Yaskawa INFORM job: X2_57-69(2)(90,180)_HARDOX.JBI

/JOB
//NAME X2_57-69(2)(90,180)_HARDOX
//POS
///NPOS 751,751,751,36,0,0
///TOOL 0
///POSTYPE PULSE
///PULSE
C00000=2000,-108350,-112464,0,80055,0
C00001=-117728,-108350,-112464,-34609,80055,-28580
C00002=-124329,53851,34766,-36826,59228,-24303
C00003=-132418,78233,54919,-18007,48363,-36393
C00004=-132091,87021,68515,-19398,44781,-35491
C00005=-131964,91219,74916,-20112,43130,-35046
C00006=-131964,92220,77875,-20603,41902,-34745
C00007=-131925,92203,77341,-20509,42211,-34802
C00008=-131397,96741,83157,-21411,41178,-34254
C00009=-131925,92203,77341,-20509,42211,-34802
C00010=-132378,78684,56627,-18262,47592,-36223
C00011=-132682,70057,46287,-17529,49367,-36706
C00012=-119143,48210,55676,-30149,44593,20608
C00013=-119357,47156,53956,-26116,42767,17551
C00014=-120340,57080,66927,-26977,39866,17985
C00015=-120719,61633,72965,-27509,38514,18256
C00016=-120718,63903,77470,-28475,37088,18806
C00017=-120500,60851,73214,-27972,38091,18544
C00018=-120914,65321,78494,-28289,37111,18678
C00019=-120500,60851,73214,-27972,38091,18544
C00020=-119122,46332,54187,-26526,42331,17820
C00021=-118999,38480,45168,-29507,46176,20252
C00022=-119368,-115903,-71302,-26914,50601,18610
C00023=-64607,-7982,-59747,18064,104585,-18556
C00024=-122585,1659,-29054,-2148,106745,-41963
C00025=-124057,3295,-23736,-2114,104277,-42416
C00026=-123367,1653,-22955,-2102,102971,-42158
C00027=-123367,1653,-22955,-2102,102971,-42158
C00028=-123367,1464,-21676,-2095,102091,-42146
C00029=-123367,1491,-21879,-2095,102231,-42148
C00030=-122595,1438,-21925,-2097,102251,-41888
C00031=-123098,1579,-22644,-2101,102754,-42066
C00032=-121099,-5117,-28172,-2107,102765,-41388
C00033=-121099,-5224,-27431,-2104,102256,-41380
C00034=-121096,-3542,-26064,-2104,102281,-41379
C00035=-121100,-4913,-29379,-2118,103615,-41403
C00036=-122679,50337,23961,-2073,99143,-41860
C00037=-122679,50327,24372,-2073,98885,-41856
C00038=-122679,50317,25468,-2068,98206,-41845
C00039=-122679,50317,25291,-2069,98316,-41847
C00040=-122229,50284,25254,-2070,98333,-41695
C00041=-122585,50333,23899,-2075,99182,-41830
C00042=-123436,20127,-8164,-2111,103367,-42191
C00043=-123085,19869,-6825,-2101,102422,-42055
C00044=-123085,19731,-5772,-2095,101704,-42044
C00045=-123090,19755,-5955,-2095,101829,-42046
C00046=-122355,19706,-6001,-2097,101852,-41798
C00047=-123021,19907,-7099,-2102,102614,-42036
C00048=-119603,42824,-10224,-2319,104332,-40939
C00049=-124323,33374,-11816,19552,90115,-11471
C00050=-119580,38024,-5833,18417,96098,-9015
C00051=-118818,47331,4592,18589,99387,-8235
C00052=-118854,51639,9991,18809,101216,-7946
C00053=-118854,51688,9891,18816,101298,-7933
C00054=-118396,53981,12432,18736,100835,-7852
C00055=-118854,51688,9891,18816,101298,-7933
C00056=-118058,50558,8647,18739,101302,-7659
C00057=-117672,49987,8022,18702,101306,-7525
C00058=-118854,52185,8952,18883,102088,-7807
C00059=-119377,80940,37276,19231,105085,60834
C00060=-119383,81426,41090,19027,103098,60507
C00061=-119383,81149,41970,18967,102452,60403
C00062=-119503,81114,41806,19281,102559,60100
C00063=-121982,78312,38330,19114,103772,59696
C00064=-119503,81115,41806,19281,102559,60100
C00065=-119566,48683,6206,18410,91622,58331
C00066=-120090,49584,7189,18533,91599,58154
C00067=-122107,80076,35944,19363,106046,60027
C00068=-125220,60788,2341,21151,116877,60889
C00069=-125220,60788,2341,21151,116877,60889
C00070=-126916,76750,29022,19801,109531,58906
C00071=-127645,78004,33974,19502,107427,58282
C00072=-127487,77220,34582,19410,106657,58208
C00073=-127487,77257,34498,19419,106724,58220
C00074=-127913,74998,31769,19485,107311,58167
C00075=-127487,77257,34498,19419,106724,58220
C00076=-124885,43382,-3109,13584,94897,56190
C00077=-125658,44980,-1455,13763,94829,55937
C00078=-126891,66473,19769,17526,104309,57625
C00079=-124484,22564,-21459,18200,86590,59420
C00080=-124478,22213,-20236,18209,85701,59290
C00081=-124478,22285,-20344,18209,85798,59305
C00082=-123939,24375,-18336,18026,85535,59441
C00083=-124479,22285,-20344,18209,85798,59305
C00084=-127548,40111,-4274,24755,95305,61297
C00085=-126910,38918,-5604,24621,95320,61520
C00086=-125531,30039,-16063,20855,91192,60400
C00087=-110493,47386,-4176,13132,86201,63779
C00088=-94830,35895,-16474,7059,86110,68517
C00089=-90477,52028,10631,17758,71006,71149
C00090=-89713,50542,11420,17514,69656,71213
C00091=-89905,50195,13035,17735,68577,70980
C00092=-89905,50233,12920,17724,68663,70994
C00093=-89883,52518,15431,17756,68305,70946
C00094=-89905,50233,12920,17724,68663,70994
C00095=-89391,49561,12188,17458,68659,71180
C00096=-88735,49652,12286,17139,68513,71391
C00097=-89905,50707,11616,17609,69662,71147
C00098=-93822,108273,63701,18536,93326,72680
C00099=-93822,107828,64715,18513,92516,72556
C00100=-93690,107878,66461,18471,91489,72445
C00101=-93690,107926,66303,18474,91606,72462
C00102=-93713,104164,61367,18504,92662,72614
C00103=-93690,107926,66303,18474,91606,72462
C00104=-88166,79692,31239,6097,86382,71862
C00105=-88845,80022,31647,6308,86349,71646
C00106=-88428,80564,30105,6176,87540,71836
C00107=-94090,77517,21608,6175,108524,71897
C00108=-94073,76835,21790,6154,108061,71879
C00109=-94073,75515,22880,6101,106718,71810
C00110=-94073,75604,22800,6105,106813,71815
C00111=-94282,72960,19602,6147,107436,71779
C00112=-94073,75604,22800,6105,106813,71815
C00113=-90523,44446,-9492,-1446,93970,71247
C00114=-91337,44548,-9384,-1199,93942,71004
C00115=-92199,55185,-1301,1007,99713,71206
C00116=-93265,18749,-25601,10213,78649,72540
C00117=-93039,18272,-23901,10154,77351,72504
C00118=-93006,18125,-22740,10166,76573,72452
C00119=-93006,18220,-22895,10161,76715,72464
C00120=-92959,20732,-20534,10144,76549,72465
C00121=-93006,18220,-22895,10161,76715,72464
C00122=-92400,18138,-22970,9886,76649,72654
C00123=-91733,17968,-23126,9585,76586,72864
C00124=-92687,19123,-24402,9968,78051,72675
C00125=-105388,2298,-39102,15529,80254,68873
C00126=-105388,1873,-38509,15552,79692,68802
C00127=-105388,1357,-37735,15585,78976,68710
C00128=-105388,1531,-38004,15573,79223,68742
C00129=-105945,-2529,-41383,15810,79315,68575
C00130=-105945,-2767,-41013,15826,78977,68531
C00131=-105742,-504,-39143,15739,78954,68594
C00132=-105548,-1447,-42806,15582,80627,68872
C00133=-86161,-6758,-47097,6979,78098,74729
C00134=-86311,-6793,-45530,7072,77135,74626
C00135=-86311,-7203,-44912,7084,76549,74590
C00136=-86311,-7084,-45095,7079,76721,74599
C00137=-86468,-10850,-48057,7154,76621,74544
C00138=-86468,-11058,-47732,7163,76316,74526
C00139=-86253,-9013,-46134,7061,76366,74599
C00140=-85946,-9538,-48533,6889,77540,74761
C00141=-91638,-28469,-60972,19623,77269,75627
C00142=-91723,-28440,-59926,19705,76695,75503
C00143=-91723,-28859,-59144,19755,76040,75393
C00144=-91723,-28693,-59463,19734,76307,75438
C00145=-94312,-27181,-58426,20833,77031,74680
C00146=-94312,-27381,-58052,20856,76717,74626
C00147=-93375,-28035,-58503,20460,76442,74902
C00148=-94102,-28107,-59801,20714,77326,74807
C00149=-75235,-25991,-61706,17727,76646,82454
C00150=-74355,-27115,-59920,17436,74870,82487
C00151=-74355,-27621,-59040,17497,74104,82374
C00152=-74355,-27526,-59211,17485,74251,82396
C00153=-73057,-27237,-59013,16875,74023,82799
C00154=-74355,-27526,-59211,17485,74251,82396
C00155=-77057,-4626,-46977,21243,91479,85327
C00156=-76984,-7096,-48960,21220,91416,85338
C00157=-74796,-23928,-59379,17950,77960,82962
C00158=-62955,11917,-39245,-2282,95516,82905
C00159=-62775,11091,-38612,-2332,94707,82971
C00160=-62775,10339,-37928,-2329,93898,82983
C00161=-62775,10494,-38073,-2330,94067,82980
C00162=-63812,9884,-38615,-2013,94064,82672
C00163=-62775,10494,-38073,-2330,94067,82980
C00164=-63124,13025,-35796,-2226,93958,82878
C00165=-62775,11512,-38975,-2336,95146,82960
C00166=-85068,-3435,-45765,9377,101067,77801
C00167=-80917,-22804,-55283,8465,96602,78792
C00168=-82338,-24881,-56282,8726,96296,78315
C00169=-82338,-25559,-54893,8703,95107,78232
C00170=-82338,-25498,-55026,8705,95219,78240
C00171=-82456,-28244,-56927,8723,94993,78185
C00172=-82338,-25498,-55026,8705,95219,78240
C00173=-82992,-25583,-55084,8828,95278,78035
C00174=-84316,-25471,-55005,9073,95425,77617
C00175=-82338,-24922,-56206,8726,96230,78312
C00176=-65428,-70038,-75520,-7958,62422,82819
C00177=-65283,-69785,-73717,-8103,61466,82944
C00178=-65283,-69734,-72466,-8160,60731,82996
C00179=-65283,-69744,-72637,-8152,60830,82990
C00180=-65562,-66708,-71125,-7963,61427,82841
C00181=-65283,-69745,-72637,-8152,60830,82990
C00182=-76204,-68518,-72352,8123,61758,80129
C00183=-74993,-68244,-72242,7504,61717,80585
C00184=-69704,-69532,-74690,-998,61942,81859
C00185=-78060,-84536,-88579,-1407,62283,78117
C00186=-78060,-84536,-88579,-1407,62283,78117
C00187=-64607,-7982,-59747,18064,104585,-18556
C00188=-43259,-142284,-94849,-68481,67043,-45987
C00189=-75789,-57542,-35879,-68380,64193,-60275
C00190=-79378,-55423,-31936,-68889,61283,-60160
C00191=-80801,-54484,-30299,-69115,60133,-60112
C00192=-80803,-53463,-27973,-69597,59790,-59668
C00193=-80780,-53792,-28606,-69479,59888,-59772
C00194=-82380,-55228,-29381,-69587,58724,-59873
C00195=-80801,-53699,-28530,-69478,59874,-59776
C00196=-81788,-51404,-27272,-69234,59369,-60118
C00197=-80801,-53699,-28530,-69478,59874,-59776
C00198=-79378,-54655,-30185,-69233,61022,-59829
C00199=-75790,-56818,-34168,-68680,63927,-59955
C00200=-84853,-69188,-42023,-59966,34850,-64425
C00201=-87616,-64026,-36454,-59770,32751,-64733
C00202=-88672,-61932,-34175,-59731,31934,-64834
C00203=-88674,-60834,-31833,-60968,31481,-64183
C00204=-88651,-60985,-32132,-60826,31549,-64256
C00205=-90372,-59623,-31443,-59618,30637,-65026
C00206=-88651,-60985,-32132,-60826,31549,-64256
C00207=-87595,-63088,-34428,-60823,32369,-64172
C00208=-84831,-68269,-40036,-60922,34477,-63902
C00209=-34135,-92769,-74242,-67244,95299,-48930
C00210=-35401,-42276,-48954,-68810,98599,-53574
C00211=-65945,-1100,7259,-69270,87048,-42040
C00212=-68239,35,11214,-69501,84806,-41537
C00213=-69159,585,12885,-69624,83908,-41331
C00214=-69161,1574,15470,-69708,83504,-40864
C00215=-69221,1430,14991,-69696,83546,-40967
C00216=-70472,2033,15498,-69808,82706,-41122
C00217=-69221,1430,14991,-69696,83546,-40967
C00218=-68301,843,13280,-69560,84443,-41175
C00219=-66008,-382,9232,-69294,86686,-41685
C00220=-65045,17742,23285,-68512,88220,-38243
C00221=-67089,19246,27753,-68708,86083,-37667
C00222=-67908,20664,31476,-68858,84932,-37105
C00223=-67909,21636,33893,-68917,84551,-36681
C00224=-67870,21286,33093,-68893,84697,-36810
C00225=-69603,21321,33122,-69077,83544,-37032
C00226=-67870,21286,33093,-68893,84697,-36810
C00227=-67052,20507,31108,-68763,85558,-37056
C00228=-65008,18839,26451,-68515,87704,-37647
C00229=-35401,-42276,-48954,-68810,98599,-53574
C00230=-34135,-92769,-74242,-67244,95299,-48930
C00231=-40047,-44089,-55446,-21687,109798,38511
C00232=-62225,-62197,-88507,-27498,109393,46828
C00233=-110162,-85165,-68253,-22495,93568,66447
C00234=-113189,-87083,-65902,-22697,90484,65921
C00235=-114452,-87710,-64890,-22792,89260,65692
C00236=-114517,-85766,-62478,-22795,88793,65757
C00237=-114452,-87710,-64890,-22792,89260,65692
C00238=-114560,-85938,-62764,-22799,88863,65728
C00239=-116855,-86136,-62847,-22980,88180,65021
C00240=-114560,-85938,-62764,-22799,88863,65728
C00241=-116037,-86901,-63721,-22918,88541,65250
C00242=-115908,-89550,-64185,-22909,87583,65481
C00243=-116037,-86901,-63721,-22918,88541,65250
C00244=-114760,-86329,-64757,-22823,89756,65485
C00245=-111694,-84556,-67168,-22619,92819,66026
C00246=-100686,-82782,-64085,-34767,78413,50947
C00247=-101124,-84756,-62575,-46086,58567,32836
C00248=-105363,-79670,-59021,-44782,56711,31479
C00249=-106963,-77579,-57544,-44243,56028,30951
C00250=-107094,-75757,-55111,-44466,55555,31127
C00251=-106963,-77579,-57544,-44243,56028,30951
C00252=-107061,-76131,-55605,-44423,55653,31093
C00253=-109164,-76621,-55827,-43839,54522,30514
C00254=-107061,-76131,-55605,-44423,55653,31093
C00255=-152521,-89404,-55591,46164,31260,-15215
C00256=-151593,-87290,-55392,44387,31486,-14209
C00257=-152521,-89404,-55591,46164,31260,-15215
C00258=-153310,-92374,-57074,47433,31236,-15946
C00259=-155515,-99823,-60624,50849,31303,-17939
C00260=-144863,-106519,-66042,48559,45403,-33907
C00261=-128223,-91539,-64179,39651,61078,-44936
C00262=-123361,-87629,-60570,38638,58731,-43541
C00263=-121491,-85978,-59075,38202,57849,-42987
C00264=-121484,-83973,-56613,38386,57460,-43144
C00265=-121491,-85978,-59075,38202,57849,-42987
C00266=-121461,-84428,-57196,38332,57549,-43096
C00267=-119429,-85653,-57392,38005,56255,-42626
C00268=-121461,-84428,-57196,38332,57549,-43096
C00269=-119967,-84308,-57809,37774,57245,-42484
C00270=-118856,-82106,-57411,37133,57477,-41844
C00271=-119967,-84308,-57809,37774,57245,-42484
C00272=-121794,-85994,-59329,38223,58099,-43033
C00273=-126552,-90004,-63001,39273,60372,-44418
C00274=-126573,-96663,-78450,37396,65213,-42514
C00275=-131304,-91681,-76533,26004,78425,-57156
C00276=-124056,-87914,-75121,11214,89260,-70181
C00277=-122142,-89367,-72002,11215,86376,-69779
C00278=-121349,-89811,-70686,11221,85247,-69607
C00279=-121343,-87912,-68316,11227,84773,-69647
C00280=-121349,-89811,-70686,11221,85247,-69607
C00281=-121327,-88115,-68626,11226,84855,-69634
C00282=-119324,-89518,-68898,11223,84034,-69016
C00283=-121327,-88115,-68626,11226,84855,-69634
C00284=-119442,-90660,-70518,11218,84452,-69019
C00285=-120607,-93154,-70984,11239,83638,-69495
C00286=-119442,-90660,-70518,11218,84452,-69019
C00287=-120261,-90277,-71864,11211,85572,-69201
C00288=-122240,-88980,-75059,11209,88432,-69628
C00289=-122263,-92131,-88871,11297,95190,-69025
C00290=-118027,-102145,-112609,-12133,81631,-15728
C00291=-114779,-111065,-98137,-30741,51344,26323
C00292=-118307,-102289,-93656,-28063,51644,24513
C00293=-119601,-98864,-91828,-27075,51783,23857
C00294=-119613,-97097,-89588,-27235,51358,23975
C00295=-119601,-98864,-91828,-27075,51783,23857
C00296=-110485,-79839,-84525,-36111,67748,27732
C00297=-112543,-80296,-84732,-35339,66815,27160
C00298=-110485,-79839,-84525,-36111,67748,27732
C00299=-133496,-108715,-92181,-7385,37609,14213
C00300=-133101,-105069,-91479,-7525,39076,14289
C00301=-133496,-108715,-92181,-7385,37609,14213
C00302=-132876,-112861,-94058,-8163,36703,14650
C00303=-131137,-123655,-98655,-10535,34221,15975
C00304=-123443,-118355,-110381,-19336,67280,34215
C00305=-114391,-92529,-101967,-29874,101827,55519
C00306=-118393,-95739,-100418,-29397,98177,54940
C00307=-120031,-96781,-99698,-29226,96757,54678
C00308=-120038,-95275,-97552,-29185,96274,54799
C00309=-120031,-96781,-99698,-29226,96757,54678
C00310=-120084,-95528,-97941,-29191,96355,54761
C00311=-122387,-95485,-97926,-29054,95580,54078
C00312=-120084,-95528,-97941,-29191,96355,54761
C00313=-120976,-97030,-99100,-29136,95998,54511
C00314=-120991,-101427,-100201,-29036,94603,54858
C00315=-120976,-97030,-99100,-29136,95998,54511
C00316=-119331,-96066,-99851,-29302,97402,54781
C00317=-115306,-93056,-101481,-29762,101015,55383
C00318=-119500,-95286,-111088,-6725,93490,23573
C00319=-126773,-109990,-105967,32242,60764,-29595
C00320=-122699,-100871,-93398,31267,56629,-29081
C00321=-121186,-97859,-91654,30361,56488,-28429
C00322=-121181,-96122,-89420,30519,56067,-28559
C00323=-121186,-97859,-91654,30361,56488,-28429
C00324=-121151,-96393,-89780,30476,56128,-28526
C00325=-118823,-96364,-89767,29286,55307,-27705
C00326=-121151,-96393,-89780,30476,56128,-28526
C00327=-120304,-96962,-90655,29967,56039,-28163
C00328=-120309,-93163,-89734,29527,57250,-27795
C00329=-120304,-96962,-90655,29967,56039,-28163
C00330=-121790,-99973,-92408,30869,56167,-28809
C00331=-125792,-107589,-96692,33228,56592,-30543
C00332=-131625,-94984,-104332,26399,91581,-50246
C00333=-126745,-145288,-119778,15495,97214,-71135
C00334=-123697,-150191,-117695,15760,92961,-70600
C00335=-122386,-151760,-116729,15896,91357,-70347
C00336=-122362,-148095,-114205,15905,91670,-70298
C00337=-122386,-151760,-116729,15896,91357,-70347
C00338=-152021,-159898,-112636,26025,88694,-79156
C00339=-148454,-161901,-113048,26644,86894,-78253
C00340=-152021,-159898,-112636,26025,88694,-79156
C00341=-97626,-122802,-108845,7114,105595,-63457
C00342=-96843,-127398,-109672,7190,103687,-63292
C00343=-97626,-122802,-108845,7114,105595,-63457
C00344=-98540,-120520,-109456,7005,107212,-63690
C00345=-100688,-114056,-110651,6782,111424,-64223
C00346=-141928,-132033,-122827,28072,87297,-56565
C00347=-127745,-107087,-104050,36954,70100,-33758
C00348=-123019,-101123,-100201,35200,68701,-32195
C00349=-121229,-98695,-98613,34495,68204,-31593
C00350=-121224,-97088,-96437,34605,67775,-31733
C00351=-121229,-98695,-98613,34495,68204,-31593
C00352=-121227,-97196,-96702,34583,67865,-31704
C00353=-118899,-97170,-96690,33712,66948,-31006
C00354=-121227,-97196,-96702,34583,67865,-31704
C00355=-120189,-96862,-97597,34041,68055,-31198
C00356=-120197,-92600,-96484,33733,69318,-30794
C00357=-120189,-96862,-97597,34041,68055,-31198
C00358=-121940,-99293,-99200,34743,68533,-31788
C00359=-126568,-105279,-103092,36497,69877,-33324
C00360=-126928,-101255,-99744,25325,80548,-44815
C00361=-122663,-98736,-96036,24420,78380,-43689
C00362=-120996,-97606,-94499,24052,77561,-43237
C00363=-120993,-95941,-92294,24092,77100,-43331
C00364=-120996,-97606,-94499,24052,77561,-43237
C00365=-121020,-96262,-92743,24089,77210,-43319
C00366=-118702,-96225,-92727,23520,76555,-42587
C00367=-121020,-96262,-92743,24089,77210,-43319
C00368=-122674,-97386,-94282,24452,78030,-43766
C00369=-126903,-99897,-97999,25343,80198,-44881
C00370=-120621,-96600,-101484,24088,62946,-45857
C00371=-120621,-96804,-99274,24394,61605,-46162
C00372=-120836,-96837,-98372,24626,61144,-46356
C00373=-120621,-96028,-104113,23676,79092,-41030
C00374=-120620,-96219,-90168,24537,71134,-42684
C00375=-106487,-107739,-103284,10074,102495,-34130
C00376=-120621,-96833,-96770,19683,109882,-37555
C00377=-120621,-96757,-99844,19967,111704,-37232
C00378=-139470,-90927,-100236,32127,92639,-54211
C00379=-120586,-139946,-100537,59993,22470,-77721
C00380=-120585,-131753,-89573,65663,21254,-80445
C00381=-120585,-129979,-87167,67023,21013,-81095
C00382=-120363,-131764,-88661,66879,20872,-81008
C00383=-120585,-129383,-86356,67491,20933,-81319
C00384=-120588,-147747,-110477,33463,48677,-59982
C00385=-120644,-140143,-100701,34547,46935,-60718
C00386=-124340,-146796,-110774,11584,101640,-53151
C00387=-120588,-147693,-110556,9391,106075,-51659
C00388=-120588,-150839,-114378,9432,106801,-51602
C00389=-120668,-127498,-127599,-8027,92338,-11843
C00390=-106540,-131828,-115388,-26739,62994,22536
C00391=-120606,-112501,-85686,-37507,17849,56930
C00392=-120605,-109780,-80480,-41231,16435,58666
C00393=-120605,-108994,-78986,-42415,16045,59215
C00394=-119980,-108543,-78089,-44300,16113,60117
C00395=-120532,-122943,-110507,-24788,69983,42881
C00396=-120328,-120551,-104070,-25274,67559,43508
C00397=-120364,-122737,-110073,-20558,99126,39146
C00398=-120608,-123337,-111674,-20610,99768,38950
C00399=-120609,-124066,-114983,-20744,101328,38677
C00400=-120610,-124421,-123392,-21260,106003,37833
C00401=-120649,-125888,-127056,-5137,96316,15534
C00402=-120651,-130620,-101533,26318,65901,-27317
C00403=-132080,-98652,-65915,40871,60604,-46715
C00404=-126739,-94814,-62411,39928,58019,-45199
C00405=-125070,-93229,-60837,39633,57144,-44743
C00406=-114661,-73601,-63122,21164,75700,-53949
C00407=-129035,-102113,-68426,24501,69140,-60716
C00408=-118965,-83311,-64570,15115,84105,-65750
C00409=-117782,-78084,-63999,13649,88678,-67245
C00410=-119873,-76495,-66852,13633,91534,-67660
C00411=-119888,-78331,-76038,13747,96118,-67156
C00412=-119081,-108028,-88031,-16388,61795,-15984
C00413=-117234,-100128,-64028,-47858,30144,31364
C00414=-117223,-96877,-58390,-50267,28944,32603
C00415=-120408,-90078,-55153,-45893,28312,30090
C00416=-121323,-87049,-53971,-43501,28942,29247
C00417=-116007,-56332,-57866,-25851,73027,43959
C00418=-110893,-121085,-68862,-33974,51532,52318
C00419=-116010,-81769,-60585,-23200,86152,63109
C00420=-116435,-73198,-57641,-22557,92556,65246
C00421=-113722,-71149,-59788,-22419,95499,65689
C00422=-113460,-61701,-78205,-24579,95746,61766
C00423=-45876,-101964,-103313,-26325,110018,55581
C00424=-15431,-40197,-19183,-56345,102197,-5038
C00425=-34862,-44642,-10243,-68104,90731,-26909
C00426=-38272,-42530,-5806,-68888,87904,-26638
C00427=-46795,4368,31406,-62110,107916,-28724
C00428=-46793,4331,31374,-62110,107918,-28724
C00429=-41809,-20527,11988,-64520,102557,-33043
C00430=-37345,-41369,-1566,-65704,98540,-31804
C00431=-38198,-39956,-806,-64837,100238,-32536
C00432=-38612,-39929,-4176,-63239,100836,-34262
C00433=-36669,-38826,-14631,-64435,105300,-36937
C00434=-35614,-75221,-31334,-66701,43579,-46020
C00435=4350,-87290,-51239,-65137,72622,-41765
C00436=-64440,-113176,-91621,-27014,43904,-67647
C00437=-122842,55452,53671,-34630,66319,4477
C00438=-122836,62423,70424,-36514,60793,6445
C00439=-123914,74645,87958,-37956,56708,7549
C00440=-124722,78954,94152,-38488,55096,7840
C00441=-125636,70258,82920,-33540,52145,4666
C00442=-125789,67542,79741,-31202,49943,1938
C00443=-125392,67161,79313,-29703,48478,313
C00444=-125087,66221,78197,-27955,47185,-1441
C00445=-124810,65557,77420,-26215,46028,-3096
C00446=-124286,65035,76747,-25175,45491,-4041
C00447=-126249,58778,70434,-20502,41712,-10718
C00448=-137325,56510,71482,20525,34338,-37678
C00449=-136832,56142,71028,20191,34313,-37446
C00450=-137859,53190,66906,20483,35518,-37713
C00451=-139227,44303,54689,20141,38626,-37648
C00452=-132675,46810,50748,-6411,52596,-1677
C00453=-131127,80601,47453,-25263,64319,-31877
C00454=-132807,97166,57058,-12495,61470,-40417
C00455=-132437,103413,60649,-12594,62499,-40395
C00456=-132694,105523,62562,-12460,62371,-40474
C00457=-135614,121161,83227,-11303,57371,-41050
C00458=-135950,123674,72731,-10332,64945,-41919
C00459=-131127,80601,47453,-25263,64319,-31877
C00460=-64440,-113176,-91621,-27014,43904,-67647
C00461=4350,-87290,-51239,-65137,72622,-41765
C00462=-52724,-99155,-43299,-70564,49554,-58260
C00463=-58609,-95164,-38578,-71970,45609,-58601
C00464=-61890,-94425,-36602,-73161,43303,-58543
C00465=-64381,-94264,-33099,-83380,35567,-51333
C00466=-59619,-87825,-31241,-79173,40525,-52280
C00467=-56306,-82378,-27652,-80427,44490,-48729
C00468=-50050,-68501,-18632,-81551,53391,-41162
C00469=-52206,-69973,-16082,-88924,49017,-35286
C00470=-51696,-72558,-17243,-91450,48356,-32919
C00471=-47167,-82165,-29359,-87907,51434,-34351
C00472=-62742,-127620,-60643,-64448,25144,-51124
C00473=-120681,-113766,-68295,-5608,40697,-75829
C00474=-94366,-50207,-56002,-165,91971,-31212
C00475=-105977,465,-13787,608,92063,-35111
C00476=-113959,39124,5892,14367,110647,55754
C00477=-126178,41136,12950,22933,109399,52257
C00478=-127720,43467,17109,22663,110067,51784
C00479=-123752,35753,9008,23415,110018,53124
C00480=-123752,35753,9008,23415,110018,53124
C00481=-130805,5914,-14980,35102,94615,48899
C00482=-123888,-16275,-33990,23627,79867,45649
C00483=-119707,-19487,-37081,14763,76374,45802
C00484=-123180,-15087,-33805,15866,77250,44700
C00485=-123180,-15087,-33805,15866,77250,44700
C00486=-117647,15650,-13979,5315,97874,47818
C00487=-127720,43467,17109,22663,110068,51784
C00488=-127474,43809,15492,22890,111084,52090
C00489=-130719,78945,34087,26234,110690,51183
C00490=-128647,79509,34777,26212,109952,51801
C00491=-129056,80436,37705,26070,110426,51724
C00492=-125584,72140,27625,26515,111148,53240
C00493=-125584,72140,27625,26515,111148,53240
C00494=-126030,64562,19391,28825,107787,52749
C00495=-124517,37218,-5406,23795,93831,49364
C00496=-123948,37834,-5518,19590,92978,48636
C00497=-123926,41560,-2510,15791,93329,47957
C00498=-123926,41560,-2510,15791,93329,47957
C00499=-124120,57245,12281,14807,101401,48035
C00500=-129056,80436,37705,26070,110426,51724
C00501=-129046,81619,36582,26323,111594,52011
C00502=-136818,40531,-19657,30108,125901,52949
C00503=-117948,36501,-23896,29804,120745,58808
C00504=-92491,72160,14210,19450,112254,63993
C00505=-88800,77970,19691,3922,110298,-90023
C00506=-93682,70864,17464,8826,106241,-90408
C00507=-92745,69457,16773,15058,105797,-88752
C00508=-92745,69457,16773,15058,105797,-88752
C00509=-91325,39794,-4644,12876,88811,-90170
C00510=-81661,24060,-16367,-6523,77566,-90489
C00511=-77455,22016,-15123,-20049,74753,-82153
C00512=-80052,21633,-15488,-18897,74199,-82956
C00513=-80052,21633,-15488,-18897,74199,-82956
C00514=-84659,40204,-4075,-10674,88037,-84920
C00515=-93682,70864,17465,8826,106241,-90408
C00516=-93725,72433,16971,8890,107342,-90340
C00517=-97940,80091,29514,9048,103156,-6949
C00518=-98908,77845,24611,16441,93303,84528
C00519=-97397,78588,31667,14482,91792,84550
C00520=-93371,76425,28694,13543,91847,85854
C00521=-93371,76425,28694,13543,91847,85854
C00522=-93768,59053,12318,15797,82985,85310
C00523=-84239,58915,12394,1180,78115,85289
C00524=-78019,74389,28829,-9380,81088,85567
C00525=-79433,76547,31257,-11066,81816,84652
C00526=-79433,76547,31257,-11066,81816,84652
C00527=-81576,92708,47930,-7426,88419,84022
C00528=-97397,78588,31667,14482,91792,84550
C00529=-97354,79703,31118,14489,92668,84667
C00530=-87269,11973,-30617,12100,94257,88059
C00531=-76731,1196,-31592,24512,84200,45976
C00532=-76093,15069,-11858,29126,84882,47191
C00533=-76496,28529,935,29255,84179,46862
C00534=-76496,28529,935,29255,84179,46862
C00535=-72773,40058,8364,20560,90031,48390
C00536=-64959,54555,20456,3747,96161,65645
C00537=-64478,47614,12836,3711,97260,65838
C00538=-65583,46047,11107,6603,100445,65963
C00539=-65583,46047,11107,6603,100445,65963
C00540=-67130,36946,2188,10743,97435,65785
C00541=-76093,15069,-11858,29126,84882,47191
C00542=-76836,15276,-13349,29279,86030,47205
C00543=-85607,4438,-25889,31272,90918,45231
C00544=-105600,-14922,-34369,38058,88899,37101
C00545=-104536,-14715,-31623,37856,87218,37002
C00546=-102074,4245,-16648,37392,86621,37853
C00547=-102074,4245,-16648,37392,86621,37853
C00548=-97922,18791,-8501,29978,95633,34790
C00549=-87110,13494,-17407,10995,92033,43188
C00550=-88395,13805,-17123,11236,92185,42780
C00551=-88656,4893,-23433,2859,86040,41268
C00552=-94618,3158,-22122,-7857,80388,37977
C00553=-94235,968,-25962,-7952,81651,38024
C00554=-104488,3284,-34697,23863,107622,43854
C00555=-109443,-2231,-31059,32377,106591,58245
C00556=-110320,-3365,-26980,32459,105627,57533
C00557=-104680,-7906,-30681,32384,103490,59158
C00558=-104680,-7906,-30681,32384,103490,59158
C00559=-104032,-32667,-47542,31839,87480,55268
C00560=-93786,-32798,-51904,17484,88289,43912
C00561=-90696,-36869,-54868,10070,85237,43878
C00562=-94885,-35577,-54035,11047,85912,42539
C00563=-94885,-35577,-54035,11047,85912,42539
C00564=-92850,-3292,-33452,7755,107506,44983
C00565=-110320,-3365,-26980,32459,105627,57533
C00566=-110385,-1906,-27994,32710,106819,57869
C00567=-118479,-29016,-58283,33773,113793,56771
C00568=-93267,-118381,-106455,-5665,75938,9980
C00569=-109157,-108939,-90497,-1929,70224,4562
C00570=-98890,-77563,-77714,-11512,91734,7109
C00571=-99855,-78102,-77961,-11450,91476,6802
C00572=-99855,-78102,-77961,-11450,91476,6802
C00573=-120192,-79065,-79185,3284,89738,-14843
C00574=-125689,-72463,-75849,6282,90924,-34709
C00575=-124219,-18600,-43381,6234,98500,-33810
C00576=-123220,42328,2705,6186,101425,-33273
C00577=-123220,42328,2705,6186,101425,-33273
C00578=-129505,65550,28545,9361,105877,-52208
C00579=-127396,78013,37963,5857,109273,-74576
C00580=-127337,81647,38799,5919,110616,-74487
C00581=-134810,-58248,-88518,5748,117553,-76769
C00582=421,-73083,-90384,-286,80877,-488
C00583=15587,-154891,-130694,-9163,4110,89788
C00584=15588,-154889,-130691,-9148,4114,89788
C00585=15588,-154889,-130691,-9148,4114,89788
C00586=14858,-154889,-130691,-11633,92017,89788
C00587=112283,-154889,-130691,-11633,92017,89788
C00588=112283,-154889,-130691,-11633,92017,89788
C00589=112283,-62920,-73826,-9987,119997,89788
C00590=112283,-102393,-124294,3297,61499,81406
C00591=116333,10372,-57760,515,78408,82890
C00592=128260,43531,-24727,-6797,75484,86129
C00593=124978,98732,43191,195,98416,85614
C00594=111986,89448,38476,5246,109507,82093
C00595=107923,82856,30204,5372,111450,-61859
C00596=107238,89541,42536,-5843,109274,-64053
C00597=106612,89158,47066,-5740,106261,-64121
C00598=106612,88915,47721,-5720,105734,-64093
C00599=106612,88944,47638,-5723,105801,-64096
C00600=106072,86499,44573,-5752,106389,-64311
C00601=106612,88944,47638,-5723,105801,-64096
C00602=107355,86213,44222,-5738,106547,-63875
C00603=107267,87282,43868,-5766,107304,-63942
C00604=109157,38294,-10767,-1770,92454,-62197
C00605=122098,33487,-9053,-25835,87636,-61879
C00606=122098,33016,-8237,-25841,86964,-61731
C00607=122098,33079,-8352,-25839,87055,-61751
C00608=121911,33071,-8361,-25782,87002,-61804
C00609=122098,33472,-9029,-25835,87615,-61873
C00610=121887,74098,33779,-25906,82606,-60850
C00611=121841,73531,35558,-25962,81341,-60588
C00612=121804,73307,36437,-25991,80739,-60468
C00613=121804,73345,36279,-25984,80844,-60491
C00614=121653,73338,36271,-25937,80797,-60537
C00615=121772,73724,34884,-25914,81783,-60712
C00616=109932,45005,-3712,-14947,87218,-62731
C00617=108690,41560,-2488,-14546,84568,-62807
C00618=108690,41213,-1926,-14554,84062,-62748
C00619=108690,41276,-2034,-14555,84157,-62760
C00620=109302,43030,-182,-14773,84030,-62545
C00621=108690,41276,-2034,-14555,84157,-62760
C00622=108322,42043,-1228,-14430,83996,-62860
C00623=107799,43213,10,-14250,83750,-63002
C00624=108690,41955,-3089,-14539,85125,-62874
C00625=122797,74033,28409,-19303,101637,-60784
C00626=123153,73032,28897,-19278,100944,-60547
C00627=123153,72589,29775,-19219,100216,-60430
C00628=123153,72658,29632,-19229,100332,-60449
C00629=122965,70214,26724,-19249,100797,-60588
C00630=123151,72891,29912,-19224,100283,-60441
C00631=125357,53352,10474,-23944,92333,-59270
C00632=124578,54201,11418,-23759,91991,-59469
C00633=123549,68107,23068,-20530,99148,-60393
C00634=139375,77155,33310,-20571,104113,-55408
C00635=139362,77177,33904,-20534,103777,-55353
C00636=139362,76787,34763,-20462,103090,-55233
C00637=139362,76841,34636,-20472,103191,-55251
C00638=139133,73828,31009,-20528,103782,-55437
C00639=139362,76841,34636,-20472,103191,-55251
C00640=140289,76211,33874,-20541,103546,-54985
C00641=140124,76528,32679,-20624,104350,-55186
C00642=138548,63755,10737,-5576,108704,40842
C00643=145128,71355,23851,3540,97913,45047
C00644=145347,72933,27344,3506,96572,45085
C00645=145347,72292,28475,3498,95548,45058
C00646=145347,72342,28378,3498,95634,45059
C00647=145165,71625,27523,3531,95796,45007
C00648=145216,72479,26693,3531,96741,45050
C00649=141877,71050,20995,10874,102520,69096
C00650=144363,74696,28515,10422,99509,69643
C00651=144363,73877,29920,10376,98243,69535
C00652=144363,73931,29819,10379,98332,69542
C00653=144258,73126,28852,10400,98523,69522
C00654=144416,74254,27504,10430,99891,69690
C00655=143755,55121,5287,15269,96239,74801
C00656=147205,61641,16125,14365,92454,75453
C00657=147205,61033,17140,14351,91548,75347
C00658=147205,61118,16990,14353,91679,75363
C00659=147489,60294,16048,14288,91784,75468
C00660=147311,60916,15198,14345,92631,75509
C00661=170235,65155,30223,8509,82624,82092
C00662=174337,65150,36108,16693,70840,83315
C00663=174322,66786,40782,16904,68890,83026
C00664=174322,66863,42245,16997,68064,82905
C00665=174322,66851,42058,16985,68169,82921
C00666=174673,63946,38689,16786,68653,83124
C00667=174322,66851,42058,16985,68169,82921
C00668=173222,65225,40168,17368,68713,82592
C00669=174109,66462,40305,16972,69056,82972
C00670=185604,29684,6830,8859,55738,85144
C00671=185703,29420,7581,8858,55135,85135
C00672=185703,29422,8629,8926,54499,85081
C00673=185703,29422,8495,8918,54579,85088
C00674=185223,31564,10625,9246,54428,84878
C00675=185703,29422,8495,8918,54579,85088
C00676=186635,31045,10103,8334,54322,85450
C00677=185698,30350,8250,8852,55205,85139
C00678=185580,32133,11274,9029,54286,85009
C00679=185580,32133,11274,9029,54286,85009
C00680=185580,32133,11274,9029,54286,85009
C00681=181189,46088,22286,19888,64756,85709
C00682=182541,68404,41066,11279,74073,86876
C00683=183780,80664,47200,4908,83799,87358
C00684=184032,88313,55510,2126,87381,81161
C00685=184032,88313,55510,2126,87381,81161
C00686=183808,73477,30884,955,87245,78265
C00687=181828,51383,11032,5786,75027,77883
C00688=185601,32078,11219,9014,54290,85018
C00689=185262,31107,8417,9098,55537,84987
C00690=174426,5329,-25167,14684,64348,81805
C00691=145128,71355,23851,3540,97913,45047
C00692=142397,69932,22654,1473,94260,56976
C00693=139251,70435,26616,12329,89216,57434
C00694=139339,71311,29404,12306,87965,57341
C00695=139306,70690,28577,12314,88153,57351
C00696=139306,70690,28577,12314,88153,57351
C00697=140509,87607,46852,9741,94560,60100
C00698=137272,97352,59900,16690,96699,66759
C00699=136078,98911,63013,20378,97423,70911
C00700=139990,81805,41480,20469,100668,72859
C00701=139990,81805,41480,20469,100668,72859
C00702=144555,63324,18895,15762,95844,78281
C00703=148294,57421,12144,9009,92386,88165
C00704=150188,63368,18949,8541,91077,88677
C00705=150188,63759,18301,8546,91669,88718
C00706=144638,48113,-4319,9997,98058,87452
C00707=138137,56114,1983,2850,104999,51664
C00708=122797,74033,28409,-19303,101637,-60784
C00709=119606,87374,42631,-13847,106662,-61571
C00710=123426,81971,35884,-14022,108645,-60408
C00711=123426,81971,35884,-14022,108645,-60408
C00712=119733,55425,4741,-4592,99836,-58987
C00713=128749,41619,-4778,-22591,89964,-58745
C00714=130269,34494,-7635,-29547,83461,-58183
C00715=127937,36021,-6073,-28734,82554,-58786
C00716=127937,36021,-6073,-28734,82554,-58786
C00717=127517,55577,11280,-29630,92933,-61673
C00718=119606,87374,42631,-13847,106662,-61571
C00719=119739,88306,42108,-13916,107461,-61620
C00720=107981,92171,45111,-5819,109093,-63790
C00721=108368,27531,-18813,-7425,80987,-75835
C00722=109501,25709,-15357,-7975,78051,-75295
C00723=105653,33535,-7574,-6352,77012,-76449
C00724=105653,33535,-7574,-6352,77012,-76449
C00725=106159,58460,13703,-8947,90525,-77595
C00726=105526,73446,29359,-8324,97975,-75777
C00727=104025,77881,33907,-1816,102433,-75339
C00728=105308,74047,29273,-1912,103343,-74930
C00729=105308,74047,29273,-1912,103343,-74930
C00730=106541,75813,31397,-4520,104649,-60328
C00731=109501,25709,-15357,-7975,78051,-75295
C00732=109312,25729,-17808,-7857,79538,-75450
C00733=104763,-5373,-51779,6205,84138,-85359
C00734=105237,-7516,-44595,6078,78614,-85484
C00735=106309,5125,-34122,5614,78593,-85145
C00736=106309,5356,-34486,5609,78934,-85129
C00737=106458,7209,-32925,5546,78916,-85084
C00738=107821,27849,-18278,3067,92181,-84630
C00739=107209,17136,-23861,5035,79502,-84863
C00740=109821,65906,27312,4040,72953,-84252
C00741=109821,66110,26707,4030,73429,-84236
C00742=110692,92621,54410,2224,80884,-83956
C00743=110645,91118,53359,2238,80760,-83973
C00744=110286,78597,43386,4214,67599,-84241
C00745=110286,79196,40601,4159,69614,-84169
C00746=111177,-64318,-84496,3679,72805,-83763
C00747=103327,-152861,-116305,9303,107136,-88261
C00748=30877,-152857,-116304,9303,107136,-88261
C00749=30877,-161292,-134334,9303,-20965,-88261
C00750=30877,-161292,-134334,9303,-20965,-88261
BC00000=30042,666204,620862
BC00001=128763,669811,393779
BC00002=128763,789553,393779
BC00003=128763,789553,268028
BC00004=128763,789553,268028
BC00005=128763,789553,268028
BC00006=128763,789553,268028
BC00007=128763,789553,268028
BC00008=128763,789553,268028
BC00009=128763,789553,268028
BC00010=128763,789553,268028
BC00011=128763,789553,268028
BC00012=117629,777144,281899
BC00013=112309,771877,272956
BC00014=112309,771877,272956
BC00015=112309,771877,272956
BC00016=112309,771877,272956
BC00017=112309,771877,272956
BC00018=112309,771877,272956
BC00019=112309,771877,272956
BC00020=112309,771877,272956
BC00021=117971,774119,541221
BC00022=117971,672934,566940
BC00023=154530,672362,58996
BC00024=300304,674227,200436
BC00025=300304,674226,200436
BC00026=300304,674226,200436
BC00027=300304,674226,200436
BC00028=300304,674226,200436
BC00029=300304,674226,200436
BC00030=300304,674226,200436
BC00031=300304,674226,200436
BC00032=300304,674226,200436
BC00033=300304,674226,200436
BC00034=300304,674226,200436
BC00035=300304,674226,200436
BC00036=300304,674226,200436
BC00037=300304,674226,200436
BC00038=300304,674226,200436
BC00039=300304,674226,200436
BC00040=300304,674226,200436
BC00041=300304,674226,200436
BC00042=300304,754989,200436
BC00043=300304,754989,200436
BC00044=300304,754989,200436
BC00045=300304,754989,200436
BC00046=300304,754989,200436
BC00047=300304,754989,200436
BC00048=300304,754989,67303
BC00049=300304,754989,67303
BC00050=300304,754989,67303
BC00051=300304,754989,67303
BC00052=300304,754989,67298
BC00053=300304,754989,67298
BC00054=300304,754989,67298
BC00055=300304,754989,67298
BC00056=300304,754989,67298
BC00057=300304,754989,67298
BC00058=300304,754989,67298
BC00059=300304,754989,67298
BC00060=300304,754989,67298
BC00061=300304,754989,67298
BC00062=300304,754989,67298
BC00063=308661,754989,67298
BC00064=300304,754989,67298
BC00065=300304,754989,67298
BC00066=300304,754989,67298
BC00067=308661,754989,48905
BC00068=308661,754989,48905
BC00069=308661,687344,48905
BC00070=308661,687344,48905
BC00071=308661,687344,48905
BC00072=308661,687344,48905
BC00073=308661,687344,48905
BC00074=308661,687344,48905
BC00075=308661,687344,48905
BC00076=308661,687344,48905
BC00077=308661,687344,48905
BC00078=308661,687344,48905
BC00079=308661,687344,48905
BC00080=308661,687344,48905
BC00081=308661,687344,48905
BC00082=308661,687344,48905
BC00083=308661,687344,48905
BC00084=308661,687344,48905
BC00085=308661,687344,48905
BC00086=308661,687344,48905
BC00087=308661,687344,48905
BC00088=283749,748214,48169
BC00089=283750,748213,48166
BC00090=283750,748213,48166
BC00091=283750,748213,48166
BC00092=283750,748213,48166
BC00093=283750,748213,48166
BC00094=283750,748213,48166
BC00095=283750,748213,48166
BC00096=283750,748213,48166
BC00097=283750,748213,48166
BC00098=283750,748213,1587
BC00099=283750,748213,1587
BC00100=283750,748213,1587
BC00101=283750,748213,1587
BC00102=283750,748213,1587
BC00103=283750,748213,1587
BC00104=283750,748213,1587
BC00105=283750,748213,1587
BC00106=283750,748213,1587
BC00107=283750,748213,1587
BC00108=283750,748213,1587
BC00109=283750,748213,1587
BC00110=283750,748213,1587
BC00111=283750,748213,1587
BC00112=283750,748213,1587
BC00113=283750,748213,1587
BC00114=283750,748213,1587
BC00115=283750,748213,1587
BC00116=283750,748213,44693
BC00117=283750,748213,44693
BC00118=283750,748213,44693
BC00119=283750,748213,44693
BC00120=283750,748213,44693
BC00121=283750,748213,44693
BC00122=283750,748213,44693
BC00123=283750,748213,44693
BC00124=283750,748213,44693
BC00125=283750,748213,44689
BC00126=283750,748213,44689
BC00127=283750,748213,44689
BC00128=283750,748213,44689
BC00129=283750,748213,44689
BC00130=283750,748213,44689
BC00131=283750,748213,44689
BC00132=283750,748213,44689
BC00133=283750,748213,44689
BC00134=283750,748213,44689
BC00135=283750,748213,44689
BC00136=283750,748213,44689
BC00137=283750,748213,44689
BC00138=283750,748213,44689
BC00139=283750,748213,44689
BC00140=283750,748213,44689
BC00141=283750,748213,44689
BC00142=283750,748213,44689
BC00143=283750,748213,44689
BC00144=283750,748213,44689
BC00145=283750,748213,44689
BC00146=283750,748213,44689
BC00147=283750,748213,44689
BC00148=283750,748213,44689
BC00149=263341,767686,31205
BC00150=263341,767686,31205
BC00151=263341,767686,31205
BC00152=263341,767686,31205
BC00153=263341,767686,31205
BC00154=263341,767686,31205
BC00155=263341,767686,31205
BC00156=263341,767686,31205
BC00157=263341,767686,31205
BC00158=263341,767686,31205
BC00159=263341,767686,31205
BC00160=263341,767686,31205
BC00161=263341,767686,31205
BC00162=263341,767686,31205
BC00163=263341,767686,31205
BC00164=263341,767686,31205
BC00165=263341,767686,31205
BC00166=263341,767686,114566
BC00167=263341,767686,114566
BC00168=263341,767686,114566
BC00169=263341,767686,114566
BC00170=263341,767686,114566
BC00171=263341,767686,114566
BC00172=263341,767686,114566
BC00173=263341,767686,114566
BC00174=263341,767686,114566
BC00175=263341,767686,114566
BC00176=263341,767686,114566
BC00177=263341,767686,114566
BC00178=263341,767686,114566
BC00179=263341,767686,114566
BC00180=263341,767686,114566
BC00181=263341,767686,114566
BC00182=263342,767686,114565
BC00183=263342,767686,114565
BC00184=263341,767686,114566
BC00185=263341,767686,114566
BC00186=259731,672693,114566
BC00187=154530,672362,58996
BC00188=398174,692224,24803
BC00189=398174,666220,198610
BC00190=398174,666220,198610
BC00191=398174,666220,198610
BC00192=398174,666220,198610
BC00193=398174,666220,198610
BC00194=398174,666220,198610
BC00195=398174,666220,198610
BC00196=398174,666220,198610
BC00197=398174,666220,198610
BC00198=398174,666220,198610
BC00199=398174,666220,198610
BC00200=398174,666220,211707
BC00201=398174,666220,211707
BC00202=398174,666220,211707
BC00203=398174,666220,211707
BC00204=398174,666220,211707
BC00205=398174,666220,211707
BC00206=398174,666220,211707
BC00207=398174,666220,211707
BC00208=398174,666220,211707
BC00209=398174,701862,55950
BC00210=398174,701862,55950
BC00211=398174,666220,226368
BC00212=398174,666220,226368
BC00213=398174,666220,226368
BC00214=398174,666220,226368
BC00215=398174,666220,226368
BC00216=398174,666220,226368
BC00217=398174,666220,226368
BC00218=398174,666220,226368
BC00219=398174,666220,226368
BC00220=398174,666220,232814
BC00221=398174,666220,232814
BC00222=398174,666220,232814
BC00223=398174,666220,232814
BC00224=398174,666220,232814
BC00225=398174,666220,232814
BC00226=398174,666220,232814
BC00227=398174,666220,232814
BC00228=398174,666220,232814
BC00229=398174,701862,55950
BC00230=398174,701862,55950
BC00231=293973,667981,1025260
BC00232=329854,694641,1042700
BC00233=398174,728005,1075175
BC00234=398174,728005,1075175
BC00235=398174,728005,1075175
BC00236=398174,728005,1075175
BC00237=398174,728005,1075175
BC00238=398174,728005,1075175
BC00239=398174,728005,1075175
BC00240=398174,728005,1075175
BC00241=398174,728005,1075175
BC00242=398174,728005,1075175
BC00243=398174,728005,1075175
BC00244=398174,728005,1075175
BC00245=398174,728005,1075175
BC00246=396804,720844,1075175
BC00247=395433,713684,1075175
BC00248=395433,713684,1075175
BC00249=395433,713684,1075175
BC00250=395433,713684,1075175
BC00251=395433,713684,1075175
BC00252=395433,713684,1075175
BC00253=395433,713684,1075175
BC00254=395433,713684,1075175
BC00255=395433,713684,1075175
BC00256=395433,713684,1075175
BC00257=395433,713684,1075175
BC00258=395433,713684,1075175
BC00259=395433,713684,1075175
BC00260=386347,707739,1075175
BC00261=377261,701795,1075175
BC00262=377261,701795,1075175
BC00263=377261,701795,1075175
BC00264=377261,701795,1075175
BC00265=377261,701795,1075175
BC00266=377261,701795,1075175
BC00267=377261,701795,1075175
BC00268=377261,701795,1075175
BC00269=377261,701795,1075175
BC00270=377261,701795,1075175
BC00271=377261,701795,1075175
BC00272=377261,701795,1075175
BC00273=377261,701795,1075175
BC00274=377261,701795,1075175
BC00275=386477,710587,1075175
BC00276=397111,720731,1075175
BC00277=397111,720731,1075175
BC00278=397111,720731,1075175
BC00279=397111,720731,1075175
BC00280=397111,720731,1075175
BC00281=397111,720731,1075175
BC00282=397111,720731,1075175
BC00283=397111,720731,1075175
BC00284=397111,720731,1075175
BC00285=397111,720731,1075175
BC00286=397111,720731,1075175
BC00287=397111,720731,1075175
BC00288=397111,720731,1075175
BC00289=397111,720731,1075175
BC00290=341550,788634,1075175
BC00291=299880,839562,1075175
BC00292=299880,839562,1075175
BC00293=299880,839562,1075175
BC00294=299880,839562,1075175
BC00295=299880,839562,1075175
BC00296=299880,839562,1075175
BC00297=299880,839562,1075175
BC00298=299880,839562,1075175
BC00299=299880,839562,1075175
BC00300=299880,839562,1075175
BC00301=299880,839562,1075175
BC00302=299880,839562,1075175
BC00303=299880,839562,1075175
BC00304=307782,859652,1075175
BC00305=316737,882421,1075175
BC00306=316737,882421,1075175
BC00307=316737,882421,1075175
BC00308=316737,882421,1075175
BC00309=316737,882421,1075175
BC00310=316737,882421,1075175
BC00311=316737,882421,1075175
BC00312=316737,882421,1075175
BC00313=316737,882421,1075175
BC00314=316737,882421,1075175
BC00315=316737,882421,1075175
BC00316=316737,882421,1075175
BC00317=316737,882421,1075175
BC00318=292135,866942,1075175
BC00319=249083,839855,1075175
BC00320=249083,839855,1075175
BC00321=249083,839855,1075175
BC00322=249083,839855,1075175
BC00323=249083,839855,1075175
BC00324=249083,839855,1075175
BC00325=249083,839855,1075175
BC00326=249083,839855,1075175
BC00327=249083,839855,1075175
BC00328=249083,839855,1075175
BC00329=249083,839855,1075175
BC00330=249083,839855,1075175
BC00331=249083,839855,1075175
BC00332=258782,860563,1075175
BC00333=268481,913400,1075175
BC00334=268481,913400,1075175
BC00335=268481,913400,1075175
BC00336=268481,913400,1075175
BC00337=268481,913400,1075175
BC00338=268481,913400,1075175
BC00339=268481,913400,1075175
BC00340=268481,913400,1075175
BC00341=268481,913400,1075175
BC00342=268481,913400,1075175
BC00343=268481,913400,1075175
BC00344=268481,913400,1075175
BC00345=268481,913400,1075175
BC00346=278935,877996,1075175
BC00347=286881,851089,1075175
BC00348=286881,851089,1075175
BC00349=286881,851089,1075175
BC00350=286881,851089,1075175
BC00351=286881,851089,1075175
BC00352=286881,851089,1075175
BC00353=286881,851089,1075175
BC00354=286881,851089,1075175
BC00355=286881,851089,1075175
BC00356=286881,851089,1075175
BC00357=286881,851089,1075175
BC00358=286881,851089,1075175
BC00359=286881,851089,1075175
BC00360=299163,799638,1075175
BC00361=299163,799638,1075175
BC00362=299163,799638,1075175
BC00363=299163,799638,1075175
BC00364=299163,799638,1075175
BC00365=299163,799638,1075175
BC00366=299163,799638,1075175
BC00367=299163,799638,1075175
BC00368=299163,799638,1075175
BC00369=299163,799638,1075175
BC00370=297700,837086,1075175
BC00371=303143,840759,1075175
BC00372=305320,842229,1075175
BC00373=302234,860773,1075175
BC00374=302039,790821,1075175
BC00375=311181,851642,1075175
BC00376=309143,852181,1075175
BC00377=304049,853528,1075175
BC00378=283572,837882,1075175
BC00379=252403,845817,1075175
BC00380=252424,845820,1075175
BC00381=257449,850758,1075175
BC00382=259459,852734,1075175
BC00383=259459,852734,1075175
BC00384=250411,880892,1075175
BC00385=250364,842699,1075175
BC00386=276234,928771,1075175
BC00387=277683,940225,1075175
BC00388=273931,944325,1075175
BC00389=280045,889701,1075175
BC00390=284292,863341,1075175
BC00391=290103,827270,1075175
BC00392=290113,827271,1075175
BC00393=285811,833355,1075175
BC00394=284091,835788,1075175
BC00395=306191,888767,1075175
BC00396=306108,858815,1075175
BC00397=300564,908599,1075175
BC00398=302671,908990,1075175
BC00399=307971,909671,1075175
BC00400=307950,909668,1075175
BC00401=326075,851507,1075175
BC00402=361001,739438,1075175
BC00403=387169,713011,1075175
BC00404=387169,713011,1075175
BC00405=387169,713011,1075175
BC00406=387169,713011,1075175
BC00407=387169,713011,1075175
BC00408=387169,713011,1075175
BC00409=387169,713011,1075175
BC00410=387169,713011,1075175
BC00411=387169,713011,1075175
BC00412=393649,712110,1075175
BC00413=397768,715690,1075175
BC00414=397768,715690,1075175
BC00415=397768,715690,1075175
BC00416=397768,715690,1075175
BC00417=397768,715690,1075175
BC00418=397768,715690,1075175
BC00419=397768,715690,1075175
BC00420=397768,715690,1075175
BC00421=397768,715690,1075175
BC00422=398174,695622,1075175
BC00423=369903,689261,936050
BC00424=391335,724220,463889
BC00425=398174,748661,291406
BC00426=398174,748661,291406
BC00427=398174,748661,291406
BC00428=398174,748661,291406
BC00429=398174,748661,291406
BC00430=398174,748661,291406
BC00431=398174,748661,291406
BC00432=398174,748661,291406
BC00433=398174,748661,291406
BC00434=398174,739157,312741
BC00435=328735,739157,312741
BC00436=38899,668753,566164
BC00437=131022,786644,300284
BC00438=131022,786644,300284
BC00439=131022,786644,300284
BC00440=131022,786644,300284
BC00441=131022,786644,300284
BC00442=131022,786644,300284
BC00443=131022,786644,300284
BC00444=131022,786644,300284
BC00445=131022,786644,300284
BC00446=131022,786644,300284
BC00447=131022,786644,300284
BC00448=131022,786644,300284
BC00449=131022,786644,300284
BC00450=131022,786644,300284
BC00451=131022,786644,300284
BC00452=135594,791682,312939
BC00453=142513,773292,255666
BC00454=135865,784786,149585
BC00455=135865,784786,97881
BC00456=135865,784786,86014
BC00457=135865,784786,86014
BC00458=135865,784786,4495
BC00459=142513,773292,255666
BC00460=38899,668753,566164
BC00461=328735,739157,312741
BC00462=368738,716608,285159
BC00463=368738,716608,285159
BC00464=368738,716608,285159
BC00465=368738,716608,285159
BC00466=368738,716608,285159
BC00467=368738,716608,285159
BC00468=368738,716608,285159
BC00469=368738,716608,285159
BC00470=368738,716608,285159
BC00471=368738,716608,285159
BC00472=369555,708134,264471
BC00473=360102,694469,304891
BC00474=265752,731081,288942
BC00475=265752,731081,288942
BC00476=279769,731080,170754
BC00477=299279,731080,170754
BC00478=299279,731080,170754
BC00479=299207,731080,171008
BC00480=299207,731080,171008
BC00481=299207,731080,171008
BC00482=299207,731080,171008
BC00483=299207,731080,171008
BC00484=299207,731080,171008
BC00485=299207,731080,171008
BC00486=299207,731080,171008
BC00487=299279,731080,170754
BC00488=299279,731080,170754
BC00489=322812,761130,32387
BC00490=323611,761129,32383
BC00491=323611,761129,32383
BC00492=323570,761079,32615
BC00493=323570,761079,32615
BC00494=323570,761079,32615
BC00495=323570,761079,61066
BC00496=323551,761056,61151
BC00497=323551,761056,61151
BC00498=323551,761056,61151
BC00499=323551,761056,61151
BC00500=323611,761129,32383
BC00501=323611,761129,32383
BC00502=323611,723724,32383
BC00503=323611,723724,32383
BC00504=275892,723724,32383
BC00505=275892,750763,16
BC00506=275964,750702,544
BC00507=275979,750690,652
BC00508=275979,750690,652
BC00509=275979,750690,56197
BC00510=275979,750691,56195
BC00511=275979,750691,56196
BC00512=275979,750691,56196
BC00513=275979,750691,56196
BC00514=275979,750691,56196
BC00515=275964,750702,544
BC00516=275964,750702,544
BC00517=307558,750702,49826
BC00518=303210,750702,14010
BC00519=303211,750702,14008
BC00520=303209,750693,14082
BC00521=303209,750693,14082
BC00522=303209,750693,14082
BC00523=289881,750693,14082
BC00524=277164,750680,14187
BC00525=277164,750680,14187
BC00526=277164,750680,14187
BC00527=277164,750680,14187
BC00528=303211,750702,14008
BC00529=303211,750702,14008
BC00530=276701,750702,115757
BC00531=243872,750702,140030
BC00532=244039,750643,140122
BC00533=244039,750643,140122
BC00534=244039,750643,140122
BC00535=244039,750643,140122
BC00536=244039,750644,140120
BC00537=244039,750644,140120
BC00538=244039,750644,140120
BC00539=244039,750644,140120
BC00540=244039,750644,140120
BC00541=244039,750643,140122
BC00542=244039,750643,140122
BC00543=244039,750643,140122
BC00544=289214,750643,152381
BC00545=289241,750591,152430
BC00546=289263,750548,152471
BC00547=289263,750548,152471
BC00548=289263,750548,152471
BC00549=289263,750548,152471
BC00550=289263,750548,152471
BC00551=289263,750548,152471
BC00552=289263,750548,152471
BC00553=289263,750548,152471
BC00554=289261,750549,152468
BC00555=289261,750549,152468
BC00556=288933,750550,152378
BC00557=288933,750550,152378
BC00558=288933,750550,152378
BC00559=288933,750550,152378
BC00560=288933,750550,152378
BC00561=288663,750551,152304
BC00562=288663,750551,152304
BC00563=288663,750551,152304
BC00564=288663,750551,152304
BC00565=288933,750550,152378
BC00566=288933,750550,152378
BC00567=288933,728871,152377
BC00568=288933,728871,152377
BC00569=288933,728871,152377
BC00570=288933,728871,152377
BC00571=288933,728871,152377
BC00572=288933,728871,152377
BC00573=288933,728871,152377
BC00574=288933,728871,152377
BC00575=288914,728880,152372
BC00576=288874,728900,100384
BC00577=288874,728900,100384
BC00578=306934,728900,100384
BC00579=313470,728900,68755
BC00580=313470,728900,68755
BC00581=313470,663693,68755
BC00582=146443,666204,652625
BC00583=204899,675147,1075138
BC00584=165935,1224131,1075137
BC00585=165935,1305468,1075137
BC00586=277861,1305468,1075137
BC00587=277861,1305468,1075137
BC00588=318353,1337579,6692
BC00589=318353,1370179,6692
BC00590=318353,1370179,6692
BC00591=318353,1370179,6692
BC00592=318353,1370179,6692
BC00593=318353,1370179,6689
BC00594=277423,1328007,56303
BC00595=277423,1328007,56303
BC00596=277423,1328007,56303
BC00597=277423,1328007,56303
BC00598=277423,1328007,56303
BC00599=277423,1328007,56303
BC00600=277423,1328007,56303
BC00601=277423,1328007,56303
BC00602=277423,1328007,56303
BC00603=277423,1328007,56303
BC00604=277423,1328007,56303
BC00605=277423,1328007,56303
BC00606=277423,1328007,56303
BC00607=277423,1328007,56303
BC00608=277423,1328007,56303
BC00609=277423,1328007,56303
BC00610=277423,1328007,56303
BC00611=277423,1328007,56303
BC00612=277423,1328007,56303
BC00613=277423,1328007,56303
BC00614=277423,1328007,56303
BC00615=277423,1328007,56303
BC00616=277423,1328007,56303
BC00617=277423,1328007,56303
BC00618=277423,1328007,56303
BC00619=277423,1328007,56303
BC00620=277423,1328007,56303
BC00621=277423,1328007,56303
BC00622=277423,1328007,56303
BC00623=277423,1328007,56303
BC00624=277423,1328007,56303
BC00625=277423,1328007,56303
BC00626=277423,1328007,56303
BC00627=277423,1328007,56303
BC00628=277423,1328007,56303
BC00629=277423,1328007,56303
BC00630=277423,1328007,56303
BC00631=277423,1328007,56303
BC00632=277423,1328007,56303
BC00633=277423,1328007,56303
BC00634=323106,1328007,56303
BC00635=323106,1328007,56303
BC00636=323106,1328007,56303
BC00637=323106,1328007,56303
BC00638=323106,1328007,56302
BC00639=323106,1328007,56303
BC00640=323106,1328007,56303
BC00641=323106,1328007,56303
BC00642=323106,1328007,56303
BC00643=323106,1328007,56303
BC00644=323106,1328007,56300
BC00645=323106,1328007,56300
BC00646=323106,1328007,56300
BC00647=323106,1328007,56300
BC00648=323106,1328007,56300
BC00649=323106,1328007,56300
BC00650=323106,1328007,56300
BC00651=323106,1328007,56300
BC00652=323106,1328007,56300
BC00653=323106,1328007,56300
BC00654=323106,1328007,56300
BC00655=323106,1328007,56300
BC00656=323106,1328007,56300
BC00657=323106,1328007,56300
BC00658=323106,1328007,56300
BC00659=323106,1328007,56300
BC00660=323106,1328007,56300
BC00661=395229,1325065,145038
BC00662=395229,1325065,145037
BC00663=395229,1325065,145037
BC00664=395229,1325065,145037
BC00665=395229,1325065,145037
BC00666=395229,1325065,145037
BC00667=395229,1325065,145037
BC00668=395229,1325065,145037
BC00669=395229,1325065,145037
BC00670=395229,1298850,145037
BC00671=395229,1298850,145037
BC00672=395229,1298850,145037
BC00673=395229,1298850,145037
BC00674=395229,1298850,145037
BC00675=395229,1298850,145037
BC00676=395229,1298850,145037
BC00677=395229,1298850,145037
BC00678=395229,1298850,145037
BC00679=395229,1298850,145037
BC00680=395229,1298850,145037
BC00681=395229,1298850,145037
BC00682=395229,1309121,145037
BC00683=395229,1309121,109272
BC00684=395229,1309121,109272
BC00685=395229,1309121,109272
BC00686=395229,1309121,57735
BC00687=395229,1309121,57735
BC00688=395229,1298850,145037
BC00689=395229,1298850,145037
BC00690=395229,1298850,145037
BC00691=323106,1328007,56303
BC00692=323106,1328007,56303
BC00693=323106,1328007,56303
BC00694=323106,1328007,56303
BC00695=323106,1328007,56303
BC00696=323106,1328007,56303
BC00697=323106,1328007,56303
BC00698=323106,1328007,56303
BC00699=323106,1328007,56303
BC00700=323106,1328007,56303
BC00701=323106,1328007,56303
BC00702=323106,1328007,56303
BC00703=323106,1328007,56303
BC00704=323106,1328007,56303
BC00705=323106,1328007,56303
BC00706=323106,1328006,56300
BC00707=323106,1328007,56302
BC00708=277423,1328007,56303
BC00709=277423,1328007,29995
BC00710=277492,1327990,30062
BC00711=277492,1327990,30062
BC00712=277492,1327990,30062
BC00713=277492,1327990,30062
BC00714=277492,1327990,30062
BC00715=277492,1327990,30062
BC00716=277492,1327990,30062
BC00717=277492,1327990,30062
BC00718=277423,1328007,29995
BC00719=277423,1328007,29995
BC00720=277423,1328007,56303
BC00721=277423,1328007,56303
BC00722=277423,1328007,56303
BC00723=277423,1328007,56268
BC00724=277423,1328007,56268
BC00725=277423,1328007,56268
BC00726=277423,1328007,56268
BC00727=277423,1328007,56202
BC00728=277423,1328007,56202
BC00729=277423,1328007,56202
BC00730=277423,1328007,56202
BC00731=277423,1328007,56303
BC00732=277423,1328007,56303
BC00733=277423,1328007,56303
BC00734=277423,1328007,56303
BC00735=277423,1328007,56303
BC00736=277423,1328007,56303
BC00737=277423,1328007,56303
BC00738=277423,1328007,56303
BC00739=277423,1328007,56303
BC00740=277423,1328007,56303
BC00741=277423,1328007,56303
BC00742=277423,1328007,56303
BC00743=277423,1328007,56303
BC00744=277423,1328007,56303
BC00745=277423,1328007,56303
BC00746=277423,1328007,56303
BC00747=277423,1328007,56303
BC00748=277423,1328006,769250
BC00749=277423,1328006,1075007
BC00750=222606,673398,1075007
EC00000=798156,1112951
EC00001=798156,1112951
EC00002=798156,1112951
EC00003=798156,1112951
EC00004=798156,1112951
EC00005=798156,1112951
EC00006=798156,1112951
EC00007=798156,1112951
EC00008=798156,1112951
EC00009=798156,1112951
EC00010=798156,1112951
EC00011=798156,1112951
EC00012=798156,1112951
EC00013=798156,1112951
EC00014=798156,1112951
EC00015=798156,1112951
EC00016=798156,1112951
EC00017=798156,1112951
EC00018=798156,1112951
EC00019=798156,1112951
EC00020=798156,1112951
EC00021=798156,1112951
EC00022=798156,1112951
EC00023=798156,1112951
EC00024=798156,1112951
EC00025=798155,1112950
EC00026=798155,1112950
EC00027=798155,1112950
EC00028=798155,1112950
EC00029=798155,1112950
EC00030=798155,1112950
EC00031=798155,1112950
EC00032=798155,1112950
EC00033=798155,1112950
EC00034=798155,1112950
EC00035=798155,1112950
EC00036=798155,1112950
EC00037=798155,1112950
EC00038=798155,1112950
EC00039=798155,1112950
EC00040=798155,1112950
EC00041=798155,1112950
EC00042=798155,1112950
EC00043=798155,1112950
EC00044=798155,1112950
EC00045=798155,1112950
EC00046=798155,1112950
EC00047=798155,1112950
EC00048=798155,1112950
EC00049=798155,1112950
EC00050=798155,1112950
EC00051=798155,1112950
EC00052=798153,1112948
EC00053=798153,1112948
EC00054=798153,1112948
EC00055=798153,1112948
EC00056=798153,1112948
EC00057=798153,1112948
EC00058=798153,1112948
EC00059=798153,1112948
EC00060=798153,1112948
EC00061=798153,1112948
EC00062=798153,1112948
EC00063=798153,1112948
EC00064=798153,1112948
EC00065=798153,1112948
EC00066=798153,1112948
EC00067=798153,1112948
EC00068=798153,1112948
EC00069=798153,1112948
EC00070=798153,1112948
EC00071=798153,1112948
EC00072=798153,1112948
EC00073=798153,1112948
EC00074=798153,1112948
EC00075=798153,1112948
EC00076=798153,1112948
EC00077=798153,1112948
EC00078=798153,1112948
EC00079=798153,1112948
EC00080=798153,1112948
EC00081=798153,1112948
EC00082=798153,1112948
EC00083=798153,1112948
EC00084=798153,1112948
EC00085=798153,1112948
EC00086=798153,1112948
EC00087=798153,1112948
EC00088=798153,1112948
EC00089=798152,1112947
EC00090=798152,1112947
EC00091=798152,1112947
EC00092=798152,1112947
EC00093=798152,1112947
EC00094=798152,1112947
EC00095=798152,1112947
EC00096=798152,1112947
EC00097=798152,1112947
EC00098=798152,1112947
EC00099=798152,1112947
EC00100=798152,1112947
EC00101=798152,1112947
EC00102=798152,1112947
EC00103=798152,1112947
EC00104=798152,1112947
EC00105=798152,1112947
EC00106=798152,1112947
EC00107=798152,1112947
EC00108=798152,1112947
EC00109=798152,1112947
EC00110=798152,1112947
EC00111=798152,1112947
EC00112=798152,1112947
EC00113=798152,1112947
EC00114=798152,1112947
EC00115=798152,1112947
EC00116=798152,1112947
EC00117=798152,1112947
EC00118=798152,1112947
EC00119=798152,1112947
EC00120=798152,1112947
EC00121=798152,1112947
EC00122=798152,1112947
EC00123=798152,1112947
EC00124=798152,1112947
EC00125=798152,1112946
EC00126=798152,1112946
EC00127=798152,1112946
EC00128=798152,1112946
EC00129=798152,1112946
EC00130=798152,1112946
EC00131=798152,1112946
EC00132=798152,1112946
EC00133=798152,1112946
EC00134=798152,1112946
EC00135=798152,1112946
EC00136=798152,1112946
EC00137=798152,1112946
EC00138=798152,1112946
EC00139=798152,1112946
EC00140=798152,1112946
EC00141=798152,1112946
EC00142=798152,1112946
EC00143=798152,1112946
EC00144=798152,1112946
EC00145=798152,1112946
EC00146=798152,1112946
EC00147=798152,1112946
EC00148=798152,1112946
EC00149=798152,1112946
EC00150=798152,1112946
EC00151=798152,1112946
EC00152=798152,1112946
EC00153=798152,1112946
EC00154=798152,1112946
EC00155=798152,1112946
EC00156=798152,1112946
EC00157=798152,1112946
EC00158=798152,1112946
EC00159=798152,1112946
EC00160=798152,1112946
EC00161=798152,1112946
EC00162=798152,1112946
EC00163=798152,1112946
EC00164=798152,1112946
EC00165=798152,1112946
EC00166=798152,1112946
EC00167=798152,1112946
EC00168=798152,1112946
EC00169=798152,1112946
EC00170=798152,1112946
EC00171=798152,1112946
EC00172=798152,1112946
EC00173=798152,1112946
EC00174=798152,1112946
EC00175=798152,1112946
EC00176=798152,1112946
EC00177=798152,1112946
EC00178=798152,1112946
EC00179=798152,1112946
EC00180=798152,1112946
EC00181=798152,1112946
EC00182=798151,1112945
EC00183=798151,1112945
EC00184=798152,1112946
EC00185=798152,1112946
EC00186=798152,1112946
EC00187=798156,1112951
EC00188=798156,1112951
EC00189=798156,1112951
EC00190=798156,1112951
EC00191=798156,1112951
EC00192=798156,1112951
EC00193=798156,1112951
EC00194=798156,1112951
EC00195=798156,1112951
EC00196=798156,1112951
EC00197=798156,1112951
EC00198=798156,1112951
EC00199=798156,1112951
EC00200=798156,1112951
EC00201=798156,1112951
EC00202=798156,1112951
EC00203=798156,1112951
EC00204=798156,1112951
EC00205=798156,1112951
EC00206=798156,1112951
EC00207=798156,1112951
EC00208=798156,1112951
EC00209=798156,1112951
EC00210=798156,1112951
EC00211=798156,1112951
EC00212=798156,1112951
EC00213=798156,1112951
EC00214=798156,1112951
EC00215=798156,1112951
EC00216=798156,1112951
EC00217=798156,1112951
EC00218=798156,1112951
EC00219=798156,1112951
EC00220=798156,1112951
EC00221=798156,1112951
EC00222=798156,1112951
EC00223=798156,1112951
EC00224=798156,1112951
EC00225=798156,1112951
EC00226=798156,1112951
EC00227=798156,1112951
EC00228=798156,1112951
EC00229=798156,1112951
EC00230=798156,1112951
EC00231=912440,1112951
EC00232=934482,1112951
EC00233=975524,1112951
EC00234=975524,1112951
EC00235=975524,1112951
EC00236=975524,1112951
EC00237=975524,1112951
EC00238=975524,1112951
EC00239=975524,1112951
EC00240=975524,1112951
EC00241=975524,1112951
EC00242=975524,1112951
EC00243=975524,1112951
EC00244=975524,1112951
EC00245=975524,1112951
EC00246=975524,1112951
EC00247=975524,1112951
EC00248=975524,1112951
EC00249=975524,1112951
EC00250=975524,1112951
EC00251=975524,1112951
EC00252=975524,1112951
EC00253=975524,1112951
EC00254=975524,1112951
EC00255=975524,1112951
EC00256=975524,1112951
EC00257=975524,1112951
EC00258=975524,1112951
EC00259=975524,1112951
EC00260=975524,1112951
EC00261=975524,1112951
EC00262=975524,1112951
EC00263=975524,1112951
EC00264=975524,1112951
EC00265=975524,1112951
EC00266=975524,1112951
EC00267=975524,1112951
EC00268=975524,1112951
EC00269=975524,1112951
EC00270=975524,1112951
EC00271=975524,1112951
EC00272=975524,1112951
EC00273=975524,1112951
EC00274=975524,1112951
EC00275=975524,1112951
EC00276=975524,1112951
EC00277=975524,1112951
EC00278=975524,1112951
EC00279=975524,1112951
EC00280=975524,1112951
EC00281=975524,1112951
EC00282=975524,1112951
EC00283=975524,1112951
EC00284=975524,1112951
EC00285=975524,1112951
EC00286=975524,1112951
EC00287=975524,1112951
EC00288=975524,1112951
EC00289=975524,1112951
EC00290=975524,1112951
EC00291=975524,1112951
EC00292=975524,1112951
EC00293=975524,1112951
EC00294=975524,1112951
EC00295=975524,1112951
EC00296=975524,1112951
EC00297=975524,1112951
EC00298=975524,1112951
EC00299=975524,1112951
EC00300=975524,1112951
EC00301=975524,1112951
EC00302=975524,1112951
EC00303=975524,1112951
EC00304=975524,1112951
EC00305=975524,1112951
EC00306=975524,1112951
EC00307=975524,1112951
EC00308=975524,1112951
EC00309=975524,1112951
EC00310=975524,1112951
EC00311=975524,1112951
EC00312=975524,1112951
EC00313=975524,1112951
EC00314=975524,1112951
EC00315=975524,1112951
EC00316=975524,1112951
EC00317=975524,1112951
EC00318=975524,1112951
EC00319=975524,1112951
EC00320=975524,1112951
EC00321=975524,1112951
EC00322=975524,1112951
EC00323=975524,1112951
EC00324=975524,1112951
EC00325=975524,1112951
EC00326=975524,1112951
EC00327=975524,1112951
EC00328=975524,1112951
EC00329=975524,1112951
EC00330=975524,1112951
EC00331=975524,1112951
EC00332=975524,1112951
EC00333=975524,1112951
EC00334=975524,1112951
EC00335=975524,1112951
EC00336=975524,1112951
EC00337=975524,1112951
EC00338=975524,1112951
EC00339=975524,1112951
EC00340=975524,1112951
EC00341=975524,1112951
EC00342=975524,1112951
EC00343=975524,1112951
EC00344=975524,1112951
EC00345=975524,1112951
EC00346=975524,1112951
EC00347=975524,1112951
EC00348=975524,1112951
EC00349=975524,1112951
EC00350=975524,1112951
EC00351=975524,1112951
EC00352=975524,1112951
EC00353=975524,1112951
EC00354=975524,1112951
EC00355=975524,1112951
EC00356=975524,1112951
EC00357=975524,1112951
EC00358=975524,1112951
EC00359=975524,1112951
EC00360=975524,1112951
EC00361=975524,1112951
EC00362=975524,1112951
EC00363=975524,1112951
EC00364=975524,1112951
EC00365=975524,1112951
EC00366=975524,1112951
EC00367=975524,1112951
EC00368=975524,1112951
EC00369=975524,1112951
EC00370=975524,1112951
EC00371=975524,1112951
EC00372=975524,1112951
EC00373=975524,1112951
EC00374=975524,1112951
EC00375=975524,1112951
EC00376=975524,1112951
EC00377=975524,1112951
EC00378=975524,1112951
EC00379=975524,1112951
EC00380=975524,1112951
EC00381=975524,1112951
EC00382=975524,1112951
EC00383=975524,1112951
EC00384=975524,1112951
EC00385=975524,1112951
EC00386=975524,1112951
EC00387=975524,1112951
EC00388=975524,1112951
EC00389=975524,1112951
EC00390=975524,1112951
EC00391=975524,1112951
EC00392=975524,1112951
EC00393=975524,1112951
EC00394=975524,1112951
EC00395=975524,1112951
EC00396=975524,1112951
EC00397=975524,1112951
EC00398=975524,1112951
EC00399=975524,1112951
EC00400=975524,1112951
EC00401=975524,1112951
EC00402=975524,1112951
EC00403=975524,1112951
EC00404=975524,1112951
EC00405=975524,1112951
EC00406=975524,1112951
EC00407=975524,1112951
EC00408=975524,1112951
EC00409=975524,1112951
EC00410=975524,1112951
EC00411=975524,1112951
EC00412=975524,1112951
EC00413=975524,1112951
EC00414=975524,1112951
EC00415=975524,1112951
EC00416=975524,1112951
EC00417=975524,1112951
EC00418=975524,1112951
EC00419=975524,1112951
EC00420=975524,1112951
EC00421=975524,1112951
EC00422=975524,1112951
EC00423=943270,1112951
EC00424=833264,1112951
EC00425=798156,1112951
EC00426=798156,1112951
EC00427=798156,1112951
EC00428=798156,1112951
EC00429=798156,1112951
EC00430=798156,1112951
EC00431=798156,1112951
EC00432=798156,1112951
EC00433=798156,1112951
EC00434=798156,1112951
EC00435=798156,1112951
EC00436=798156,1112951
EC00437=798156,1112951
EC00438=798156,1112951
EC00439=798156,1112951
EC00440=798156,1112951
EC00441=798156,1112951
EC00442=798156,1112951
EC00443=798156,1112951
EC00444=798156,1112951
EC00445=798156,1112951
EC00446=798156,1112951
EC00447=798156,1112951
EC00448=798156,1112951
EC00449=798156,1112951
EC00450=798156,1112951
EC00451=798156,1112951
EC00452=798156,1112951
EC00453=798156,1112951
EC00454=798156,1112951
EC00455=798156,1112951
EC00456=798156,1112951
EC00457=798156,1112951
EC00458=798156,1112951
EC00459=798156,1112951
EC00460=798156,1112951
EC00461=798156,1112951
EC00462=798156,1112951
EC00463=798156,1112951
EC00464=798156,1112951
EC00465=798156,1112951
EC00466=798156,1112951
EC00467=798156,1112951
EC00468=798156,1112951
EC00469=798156,1112951
EC00470=798156,1112951
EC00471=798156,1112951
EC00472=798156,1112951
EC00473=798156,1112951
EC00474=798156,1112951
EC00475=798156,1112951
EC00476=798155,1112950
EC00477=798155,1112950
EC00478=798155,1112950
EC00479=798155,1112950
EC00480=798155,1112950
EC00481=798155,1112950
EC00482=798155,1112950
EC00483=798155,1112950
EC00484=798155,1112950
EC00485=798155,1112950
EC00486=798155,1112950
EC00487=798155,1112950
EC00488=798155,1112950
EC00489=798155,1112950
EC00490=798154,1112949
EC00491=798154,1112949
EC00492=798154,1112949
EC00493=798154,1112949
EC00494=798154,1112949
EC00495=798154,1112949
EC00496=798154,1112949
EC00497=798154,1112949
EC00498=798154,1112949
EC00499=798154,1112949
EC00500=798154,1112949
EC00501=798154,1112949
EC00502=798154,1112949
EC00503=798154,1112949
EC00504=798154,1112949
EC00505=798153,1112948
EC00506=798153,1112948
EC00507=798153,1112948
EC00508=798153,1112948
EC00509=798153,1112948
EC00510=798152,1112946
EC00511=798152,1112946
EC00512=798152,1112946
EC00513=798152,1112946
EC00514=798152,1112946
EC00515=798153,1112948
EC00516=798153,1112948
EC00517=798153,1112948
EC00518=798152,1112946
EC00519=798151,1112944
EC00520=798151,1112944
EC00521=798151,1112944
EC00522=798151,1112944
EC00523=798151,1112944
EC00524=798151,1112944
EC00525=798151,1112944
EC00526=798151,1112944
EC00527=798151,1112944
EC00528=798151,1112944
EC00529=798151,1112944
EC00530=798151,1112943
EC00531=798151,1112943
EC00532=798150,1112942
EC00533=798150,1112942
EC00534=798150,1112942
EC00535=798150,1112942
EC00536=798148,1112939
EC00537=798148,1112939
EC00538=798148,1112939
EC00539=798148,1112939
EC00540=798148,1112939
EC00541=798150,1112942
EC00542=798150,1112942
EC00543=798150,1112942
EC00544=798150,1112942
EC00545=798150,1112942
EC00546=798150,1112942
EC00547=798150,1112942
EC00548=798150,1112942
EC00549=798150,1112942
EC00550=798150,1112942
EC00551=798150,1112942
EC00552=798150,1112942
EC00553=798150,1112942
EC00554=798149,1112940
EC00555=798149,1112940
EC00556=798149,1112940
EC00557=798149,1112940
EC00558=798149,1112940
EC00559=798149,1112940
EC00560=798149,1112940
EC00561=798149,1112940
EC00562=798149,1112940
EC00563=798149,1112940
EC00564=798149,1112940
EC00565=798149,1112940
EC00566=798149,1112940
EC00567=798148,1112939
EC00568=798148,1112939
EC00569=798148,1112939
EC00570=798148,1112939
EC00571=798148,1112939
EC00572=798148,1112939
EC00573=798148,1112939
EC00574=798148,1112939
EC00575=798148,1112939
EC00576=798148,1112939
EC00577=798148,1112939
EC00578=798148,1112939
EC00579=798148,1112939
EC00580=798148,1112939
EC00581=798148,1112939
EC00582=798156,1112951
EC00583=798152,1112946
EC00584=798151,1112945
EC00585=798151,1112945
EC00586=798151,1112945
EC00587=798151,1112945
EC00588=798151,1112945
EC00589=798151,1112945
EC00590=798151,1112945
EC00591=798151,1112945
EC00592=798151,1112945
EC00593=798136,1112931
EC00594=798136,1112931
EC00595=798136,1112931
EC00596=798136,1112931
EC00597=798136,1112931
EC00598=798136,1112931
EC00599=798136,1112931
EC00600=798136,1112931
EC00601=798136,1112931
EC00602=798136,1112931
EC00603=798136,1112931
EC00604=798136,1112931
EC00605=798136,1112931
EC00606=798136,1112931
EC00607=798136,1112931
EC00608=798136,1112931
EC00609=798136,1112931
EC00610=798136,1112931
EC00611=798136,1112931
EC00612=798136,1112931
EC00613=798136,1112931
EC00614=798136,1112931
EC00615=798136,1112931
EC00616=798136,1112931
EC00617=798136,1112931
EC00618=798136,1112931
EC00619=798136,1112931
EC00620=798136,1112931
EC00621=798136,1112931
EC00622=798136,1112931
EC00623=798136,1112931
EC00624=798136,1112931
EC00625=798136,1112931
EC00626=798136,1112931
EC00627=798136,1112931
EC00628=798136,1112931
EC00629=798136,1112931
EC00630=798136,1112931
EC00631=798136,1112931
EC00632=798136,1112931
EC00633=798136,1112931
EC00634=798136,1112931
EC00635=798136,1112931
EC00636=798136,1112931
EC00637=798136,1112931
EC00638=798136,1112930
EC00639=798136,1112931
EC00640=798136,1112931
EC00641=798136,1112931
EC00642=798136,1112931
EC00643=798136,1112931
EC00644=798136,1112931
EC00645=798136,1112931
EC00646=798136,1112931
EC00647=798136,1112931
EC00648=798136,1112931
EC00649=798136,1112931
EC00650=798136,1112931
EC00651=798136,1112931
EC00652=798136,1112931
EC00653=798136,1112931
EC00654=798136,1112931
EC00655=798136,1112931
EC00656=798136,1112931
EC00657=798136,1112931
EC00658=798136,1112931
EC00659=798136,1112931
EC00660=798136,1112931
EC00661=798135,1112930
EC00662=798134,1112929
EC00663=798134,1112929
EC00664=798134,1112929
EC00665=798134,1112929
EC00666=798134,1112929
EC00667=798134,1112929
EC00668=798134,1112929
EC00669=798134,1112929
EC00670=798134,1112929
EC00671=798134,1112929
EC00672=798134,1112929
EC00673=798134,1112929
EC00674=798134,1112929
EC00675=798134,1112929
EC00676=798134,1112929
EC00677=798134,1112929
EC00678=798134,1112929
EC00679=798134,1112929
EC00680=798134,1112929
EC00681=798134,1112929
EC00682=798134,1112929
EC00683=798134,1112929
EC00684=798134,1112929
EC00685=798134,1112929
EC00686=798134,1112929
EC00687=798134,1112929
EC00688=798134,1112929
EC00689=798134,1112929
EC00690=798134,1112929
EC00691=798136,1112931
EC00692=798136,1112931
EC00693=798136,1112931
EC00694=798136,1112931
EC00695=798136,1112931
EC00696=798136,1112931
EC00697=798136,1112931
EC00698=798136,1112931
EC00699=798136,1112931
EC00700=798136,1112931
EC00701=798136,1112931
EC00702=798136,1112931
EC00703=798136,1112931
EC00704=798136,1112931
EC00705=798136,1112931
EC00706=798135,1112929
EC00707=798135,1112930
EC00708=798136,1112931
EC00709=798136,1112931
EC00710=798136,1112931
EC00711=798136,1112931
EC00712=798136,1112931
EC00713=798136,1112931
EC00714=798136,1112931
EC00715=798136,1112931
EC00716=798136,1112931
EC00717=798136,1112931
EC00718=798136,1112931
EC00719=798136,1112931
EC00720=798136,1112931
EC00721=798136,1112931
EC00722=798136,1112931
EC00723=798136,1112931
EC00724=798136,1112931
EC00725=798136,1112931
EC00726=798136,1112931
EC00727=798136,1112931
EC00728=798136,1112931
EC00729=798136,1112931
EC00730=798136,1112931
EC00731=798136,1112931
EC00732=798136,1112931
EC00733=798136,1112931
EC00734=798136,1112931
EC00735=798136,1112931
EC00736=798136,1112931
EC00737=798136,1112931
EC00738=798136,1112931
EC00739=798136,1112931
EC00740=798136,1112931
EC00741=798136,1112931
EC00742=798136,1112931
EC00743=798136,1112931
EC00744=798136,1112931
EC00745=798136,1112931
EC00746=798136,1112931
EC00747=798136,1112931
EC00748=798135,1112930
EC00749=798135,1112929
EC00750=798135,1112929
///POSTYPE BASE
///RECTAN
///RCONF 0,0,0,0,0,0,0,0,0,0,0,0,0,0,0,0,0,0,0,0,0,0,0,0
P00006=0.222,-3.123,-1.508,0.0000,0.0000,0.0000
P00020=2.715,4.999,8.452,0.0000,0.0000,0.0000
P00022=0.222,-3.123,-1.508,0.0000,0.0000,0.0000
P00023=0.143,-0.036,0.682,0.0000,0.0000,0.0000
P00024=0.145,-0.552,1.326,0.0000,0.0000,0.0000
P00025=-2.003,0.006,0.728,0.0000,0.0000,0.0000
P00026=0.562,-0.002,-0.337,0.0000,0.0000,0.0000
P00031=1.853,-0.001,-1.549,0.0000,0.0000,0.0000
P00032=1.957,0.503,-7.217,0.0000,0.0000,0.0000
///RCONF 0,0,0,0,1,0,0,0,0,0,0,0,0,0,0,0,0,0,0,0,0,0,0,0
P00033=-0.123,0.612,-5.012,0.0000,0.0000,0.0000
///RCONF 0,0,0,0,0,0,0,0,0,0,0,0,0,0,0,0,0,0,0,0,0,0,0,0
P00034=-0.304,0.773,-2.693,0.0000,0.0000,0.0000
P00035=2.817,0.591,-1.622,0.0000,0.0000,0.0000
P00036=-1.108,-0.829,1.850,0.0000,0.0000,0.0000
P00037=0.023,0.937,-2.677,0.0000,0.0000,0.0000
P00038=0.158,-1.133,-1.952,0.0000,0.0000,0.0000
P00039=0.012,-3.081,-0.106,0.0000,0.0000,0.0000
P00040=-0.030,9.648,2.467,0.0000,0.0000,0.0000
P00050=4.296,-4.501,-0.826,0.0000,0.0000,0.0000
P00051=0.367,3.892,0.009,0.0000,0.0000,0.0000
P00052=0.088,2.832,-0.342,0.0000,0.0000,0.0000
P00053=0.134,6.594,0.107,0.0000,0.0000,0.0000
P00054=-0.103,6.509,-0.702,0.0000,0.0000,0.0000
P00055=-0.342,8.912,1.324,0.0000,0.0000,0.0000
P00056=0.568,-0.032,0.830,0.0000,0.0000,0.0000
P00057=0.586,-0.180,1.727,0.0000,0.0000,0.0000
P00058=0.385,-0.061,1.027,0.0000,0.0000,0.0000
P00059=0.483,-0.984,-2.888,0.0000,0.0000,0.0000
P00060=2.327,-2.514,-2.692,0.0000,0.0000,0.0000
P00061=1.575,-3.405,-0.752,0.0000,0.0000,0.0000
P00062=-0.135,-0.848,-1.706,0.0000,0.0000,0.0000
P00063=0.036,-0.654,-3.005,0.0000,0.0000,0.0000
P00064=-0.056,-0.423,-1.596,0.0000,0.0000,0.0000
P00065=-5.731,-1.657,0.588,0.0000,0.0000,0.0000
P00070=0.003,2.805,-1.116,0.0000,0.0000,0.0000
P00071=2.716,0.070,1.352,0.0000,0.0000,0.0000
P00072=1.041,-0.003,-0.797,0.0000,0.0000,0.0000
//INST
///DATE 2025/03/13 09:59
///ATTR SC,RW
///GROUP1 RB1,BS1
///GROUP2 ST1
NOP
'X2_57-69(2)(90,180)
'Down
MOVJ C00000 BC00000 VJ=100.00  +MOVJ EC00000 VJ=100.00
MOVJ C00001 BC00001 VJ=100.00  +MOVJ EC00001 VJ=100.00
MOVJ C00002 BC00002 VJ=100.00  +MOVJ EC00002 VJ=100.00
'Path S4549
SFTOF3D
MOVJ C00003 BC00003 VJ=100.00  +MOVJ EC00003 VJ=100.00
MOVL C00004 BC00004 V=800.0  +MOVJ EC00004 VJ=100.00
SMOVL C00005 BC00005 V=166.7  +MOVJ EC00005
SREFP 3 C00006 BC00006  +REFP EC00006
CALL JOB:SEARCH-R1-S13D
SET P020 P006
SFTON3D P020
SMOVL C00007 BC00007 V=166.7  +MOVJ EC00007
SREFP 3 C00008 BC00008  +REFP EC00008
CALL JOB:SEARCH-R1-S13D
SET P020 P006
SFTON3D P020
SMOVL C00009 BC00009 V=166.7  +MOVJ EC00009
MOVL C00010 BC00010 V=1000.0  +MOVJ EC00010 VJ=100.00
'EndPath S4549
'Path S3846
SFTOF3D
MOVJ C00011 BC00011 VJ=100.00  +MOVJ EC00011 VJ=100.00
MOVJ C00012 BC00012 VJ=100.00  +MOVJ EC00012 VJ=100.00
'EndPath S3846
'Path S4550
SFTOF3D
MOVJ C00013 BC00013 VJ=100.00  +MOVJ EC00013 VJ=100.00
MOVL C00014 BC00014 V=800.0  +MOVJ EC00014 VJ=100.00
SMOVL C00015 BC00015 V=166.7  +MOVJ EC00015
SREFP 3 C00016 BC00016  +REFP EC00016
CALL JOB:SEARCH-R1-S13D
SET P022 P006
SFTON3D P022
SMOVL C00017 BC00017 V=166.7  +MOVJ EC00017
SREFP 3 C00018 BC00018  +REFP EC00018
CALL JOB:SEARCH-R1-S13D
SET P022 P006
SFTON3D P022
SMOVL C00019 BC00019 V=166.7  +MOVJ EC00019
MOVL C00020 BC00020 V=1000.0  +MOVJ EC00020 VJ=100.00
'EndPath S4550
MOVJ C00021 BC00021 VJ=100.00  +MOVJ EC00021 VJ=100.00
MOVJ C00022 BC00022 VJ=100.00  +MOVJ EC00022 VJ=100.00
MOVJ C00023 BC00023 VJ=100.00  +MOVJ EC00023 VJ=100.00
'Path S4663
SFTOF3D
MOVJ C00024 BC00024 VJ=100.00  +MOVJ EC00024 VJ=100.00
MOVL C00025 BC00025 V=800.0  +MOVJ EC00025 VJ=100.00
SMOVL C00026 BC00026 V=166.7  +MOVJ EC00026
SMOVL C00027 BC00027 V=166.7  +MOVJ EC00027
SREFP 3 C00028 BC00028  +REFP EC00028
CALL JOB:SEARCH-R1-S13D
SET P051 P006
SFTON3D P051
SMOVL C00029 BC00029 V=166.7  +MOVJ EC00029
SREFP 3 C00030 BC00030  +REFP EC00030
CALL JOB:SEARCH-R1-S13D
SET P051 P006
SFTON3D P051
SMOVL C00031 BC00031 V=166.7  +MOVJ EC00031
SMOVL C00032 BC00032 V=166.7  +MOVJ EC00032
SMOVL C00033 BC00033 V=166.7  +MOVJ EC00033
SREFP 3 C00034 BC00034  +REFP EC00034
CALL JOB:SEARCH-R1-S13D
SET P051 P006
SFTON3D P051
SMOVL C00035 BC00035 V=166.7  +MOVJ EC00035
SFTOF3D
MOVL C00036 BC00036 V=800.0  +MOVJ EC00036 VJ=100.00
SMOVL C00037 BC00037 V=166.7  +MOVJ EC00037
SREFP 3 C00038 BC00038  +REFP EC00038
CALL JOB:SEARCH-R1-S13D
SET P052 P006
SFTON3D P052
SMOVL C00039 BC00039 V=166.7  +MOVJ EC00039
SREFP 3 C00040 BC00040  +REFP EC00040
CALL JOB:SEARCH-R1-S13D
SET P052 P006
SFTON3D P052
SMOVL C00041 BC00041 V=166.7  +MOVJ EC00041
SFTOF3D
MOVL C00042 BC00042 V=800.0  +MOVJ EC00042 VJ=100.00
SMOVL C00043 BC00043 V=166.7  +MOVJ EC00043
SREFP 3 C00044 BC00044  +REFP EC00044
CALL JOB:SEARCH-R1-S13D
SET P053 P006
SFTON3D P053
SMOVL C00045 BC00045 V=166.7  +MOVJ EC00045
SREFP 3 C00046 BC00046  +REFP EC00046
CALL JOB:SEARCH-R1-S13D
SET P053 P006
SFTON3D P053
SMOVL C00047 BC00047 V=166.7  +MOVJ EC00047
MOVJ C00048 BC00048 VJ=100.00  +MOVJ EC00048 VJ=100.00
MOVJ C00049 BC00049 VJ=100.00  +MOVJ EC00049 VJ=100.00
MOVL C00050 BC00050 V=333.3  +MOVJ EC00050 VJ=100.00
MOVL C00051 BC00051 V=166.7  +MOVJ EC00051 VJ=100.00
SREFP 3 C00052 BC00052  +REFP EC00052
CALL JOB:SEARCH-R1-S13D
SET P055 P006
SFTON3D P055
SMOVL C00053 BC00053 V=166.7  +MOVJ EC00053
SREFP 3 C00054 BC00054  +REFP EC00054
CALL JOB:SEARCH-R1-S13D
SET P055 P006
SFTON3D P055
SMOVL C00055 BC00055 V=166.7  +MOVJ EC00055
SMOVL C00056 BC00056 V=166.7  +MOVJ EC00056
SREFP 3 C00057 BC00057  +REFP EC00057
CALL JOB:SEARCH-R1-S13D
SET P055 P006
SFTON3D P055
SMOVL C00058 BC00058 V=166.7  +MOVJ EC00058
MOVJ C00059 BC00059 VJ=100.00  +MOVJ EC00059 VJ=100.00
MOVL C00060 BC00060 V=166.7  +MOVJ EC00060 VJ=100.00
SREFP 3 C00061 BC00061  +REFP EC00061
CALL JOB:SEARCH-R1-S13D
SET P054 P006
SFTON3D P054
SMOVL C00062 BC00062 V=166.7  +MOVJ EC00062
SREFP 3 C00063 BC00063  +REFP EC00063
CALL JOB:SEARCH-R1-S13D
SET P054 P006
SFTON3D P054
SMOVL C00064 BC00064 V=166.7  +MOVJ EC00064
SMOVL C00065 BC00065 V=166.7  +MOVJ EC00065
SREFP 3 C00066 BC00066  +REFP EC00066
CALL JOB:SEARCH-R1-S13D
SET P054 P006
SFTON3D P054
SMOVL C00067 BC00067 V=166.7  +MOVJ EC00067
SMOVL C00068 BC00068 V=666.7  +MOVJ EC00068
MOVL C00069 BC00069 V=666.7  +MOVJ EC00069 VJ=100.00
MOVL C00070 BC00070 V=666.7  +MOVJ EC00070 VJ=100.00
MOVL C00071 BC00071 V=166.7  +MOVJ EC00071 VJ=100.00
SREFP 3 C00072 BC00072  +REFP EC00072
CALL JOB:SEARCH-R1-S13D
SET P056 P006
SFTON3D P056
SMOVL C00073 BC00073 V=166.7  +MOVJ EC00073
SREFP 3 C00074 BC00074  +REFP EC00074
CALL JOB:SEARCH-R1-S13D
SET P056 P006
SFTON3D P056
SMOVL C00075 BC00075 V=166.7  +MOVJ EC00075
SMOVL C00076 BC00076 V=166.7  +MOVJ EC00076
SREFP 3 C00077 BC00077  +REFP EC00077
CALL JOB:SEARCH-R1-S13D
SET P056 P006
SFTON3D P056
SMOVL C00078 BC00078 V=166.7  +MOVJ EC00078
MOVL C00079 BC00079 V=166.7  +MOVJ EC00079 VJ=100.00
SREFP 3 C00080 BC00080  +REFP EC00080
CALL JOB:SEARCH-R1-S13D
SET P057 P006
SFTON3D P057
SMOVL C00081 BC00081 V=166.7  +MOVJ EC00081
SREFP 3 C00082 BC00082  +REFP EC00082
CALL JOB:SEARCH-R1-S13D
SET P057 P006
SFTON3D P057
SMOVL C00083 BC00083 V=166.7  +MOVJ EC00083
SMOVL C00084 BC00084 V=166.7  +MOVJ EC00084
SREFP 3 C00085 BC00085  +REFP EC00085
CALL JOB:SEARCH-R1-S13D
SET P057 P006
SFTON3D P057
SMOVL C00086 BC00086 V=166.7  +MOVJ EC00086
MOVL C00087 BC00087 V=666.7  +MOVJ EC00087 VJ=100.00
MOVL C00088 BC00088 V=666.7  +MOVJ EC00088 VJ=100.00
MOVL C00089 BC00089 V=666.7  +MOVJ EC00089 VJ=100.00
MOVL C00090 BC00090 V=166.7  +MOVJ EC00090 VJ=100.00
SREFP 3 C00091 BC00091  +REFP EC00091
CALL JOB:SEARCH-R1-S13D
SET P058 P006
SFTON3D P058
SMOVL C00092 BC00092 V=166.7  +MOVJ EC00092
SREFP 3 C00093 BC00093  +REFP EC00093
CALL JOB:SEARCH-R1-S13D
SET P058 P006
SFTON3D P058
SMOVL C00094 BC00094 V=166.7  +MOVJ EC00094
SMOVL C00095 BC00095 V=166.7  +MOVJ EC00095
SREFP 3 C00096 BC00096  +REFP EC00096
CALL JOB:SEARCH-R1-S13D
SET P058 P006
SFTON3D P058
SMOVL C00097 BC00097 V=166.7  +MOVJ EC00097
MOVL C00098 BC00098 V=666.7  +MOVJ EC00098 VJ=100.00
MOVL C00099 BC00099 V=166.7  +MOVJ EC00099 VJ=100.00
SREFP 3 C00100 BC00100  +REFP EC00100
CALL JOB:SEARCH-R1-S13D
SET P059 P006
SFTON3D P059
SMOVL C00101 BC00101 V=166.7  +MOVJ EC00101
SREFP 3 C00102 BC00102  +REFP EC00102
CALL JOB:SEARCH-R1-S13D
SET P059 P006
SFTON3D P059
SMOVL C00103 BC00103 V=166.7  +MOVJ EC00103
SMOVL C00104 BC00104 V=166.7  +MOVJ EC00104
SREFP 3 C00105 BC00105  +REFP EC00105
CALL JOB:SEARCH-R1-S13D
SET P059 P006
SFTON3D P059
SMOVL C00106 BC00106 V=166.7  +MOVJ EC00106
MOVL C00107 BC00107 V=666.7  +MOVJ EC00107 VJ=100.00
MOVL C00108 BC00108 V=166.7  +MOVJ EC00108 VJ=100.00
SREFP 3 C00109 BC00109  +REFP EC00109
CALL JOB:SEARCH-R1-S13D
SET P060 P006
SFTON3D P060
SMOVL C00110 BC00110 V=166.7  +MOVJ EC00110
SREFP 3 C00111 BC00111  +REFP EC00111
CALL JOB:SEARCH-R1-S13D
SET P060 P006
SFTON3D P060
SMOVL C00112 BC00112 V=166.7  +MOVJ EC00112
SMOVL C00113 BC00113 V=166.7  +MOVJ EC00113
SREFP 3 C00114 BC00114  +REFP EC00114
CALL JOB:SEARCH-R1-S13D
SET P060 P006
SFTON3D P060
SMOVL C00115 BC00115 V=166.7  +MOVJ EC00115
MOVL C00116 BC00116 V=666.7  +MOVJ EC00116 VJ=100.00
MOVL C00117 BC00117 V=166.7  +MOVJ EC00117 VJ=100.00
SREFP 3 C00118 BC00118  +REFP EC00118
CALL JOB:SEARCH-R1-S13D
SET P061 P006
SFTON3D P061
SMOVL C00119 BC00119 V=166.7  +MOVJ EC00119
SREFP 3 C00120 BC00120  +REFP EC00120
CALL JOB:SEARCH-R1-S13D
SET P061 P006
SFTON3D P061
SMOVL C00121 BC00121 V=166.7  +MOVJ EC00121
SMOVL C00122 BC00122 V=166.7  +MOVJ EC00122
SREFP 3 C00123 BC00123  +REFP EC00123
CALL JOB:SEARCH-R1-S13D
SET P061 P006
SFTON3D P061
SMOVL C00124 BC00124 V=166.7  +MOVJ EC00124
MOVL C00125 BC00125 V=666.7  +MOVJ EC00125 VJ=100.00
MOVL C00126 BC00126 V=166.7  +MOVJ EC00126 VJ=100.00
SREFP 3 C00127 BC00127  +REFP EC00127
CALL JOB:SEARCH-R1-S13D
SET P070 P006
SFTON3D P070
SMOVL C00128 BC00128 V=166.7  +MOVJ EC00128
MOVL C00129 BC00129 V=166.7  +MOVJ EC00129 VJ=100.00
MOVL C00130 BC00130 V=166.7  +MOVJ EC00130 VJ=100.00
SREFP 3 C00131 BC00131  +REFP EC00131
CALL JOB:SEARCH-R1-S13D
SET P070 P006
SFTON3D P070
SMOVL C00132 BC00132 V=166.7  +MOVJ EC00132
SFTOF3D
MOVL C00133 BC00133 V=666.7  +MOVJ EC00133 VJ=100.00
MOVL C00134 BC00134 V=166.7  +MOVJ EC00134 VJ=100.00
SREFP 3 C00135 BC00135  +REFP EC00135
CALL JOB:SEARCH-R1-S13D
SET P071 P006
SFTON3D P071
SMOVL C00136 BC00136 V=166.7  +MOVJ EC00136
MOVL C00137 BC00137 V=166.7  +MOVJ EC00137 VJ=100.00
MOVL C00138 BC00138 V=166.7  +MOVJ EC00138 VJ=100.00
SREFP 3 C00139 BC00139  +REFP EC00139
CALL JOB:SEARCH-R1-S13D
SET P071 P006
SFTON3D P071
SMOVL C00140 BC00140 V=166.7  +MOVJ EC00140
SFTOF3D
MOVL C00141 BC00141 V=666.7  +MOVJ EC00141 VJ=100.00
MOVL C00142 BC00142 V=166.7  +MOVJ EC00142 VJ=100.00
SREFP 3 C00143 BC00143  +REFP EC00143
CALL JOB:SEARCH-R1-S13D
SET P072 P006
SFTON3D P072
SMOVL C00144 BC00144 V=166.7  +MOVJ EC00144
MOVL C00145 BC00145 V=166.7  +MOVJ EC00145 VJ=100.00
MOVL C00146 BC00146 V=166.7  +MOVJ EC00146 VJ=100.00
SREFP 3 C00147 BC00147  +REFP EC00147
CALL JOB:SEARCH-R1-S13D
SET P072 P006
SFTON3D P072
SMOVL C00148 BC00148 V=166.7  +MOVJ EC00148
MOVL C00149 BC00149 V=666.7  +MOVJ EC00149 VJ=100.00
MOVL C00150 BC00150 V=166.7  +MOVJ EC00150 VJ=100.00
SREFP 3 C00151 BC00151  +REFP EC00151
CALL JOB:SEARCH-R1-S13D
SET P063 P006
SFTON3D P063
SMOVL C00152 BC00152 V=166.7  +MOVJ EC00152
SREFP 3 C00153 BC00153  +REFP EC00153
CALL JOB:SEARCH-R1-S13D
SET P063 P006
SFTON3D P063
SMOVL C00154 BC00154 V=166.7  +MOVJ EC00154
SMOVL C00155 BC00155 V=166.7  +MOVJ EC00155
SREFP 3 C00156 BC00156  +REFP EC00156
CALL JOB:SEARCH-R1-S13D
SET P063 P006
SFTON3D P063
SMOVL C00157 BC00157 V=166.7  +MOVJ EC00157
MOVL C00158 BC00158 V=666.7  +MOVJ EC00158 VJ=100.00
MOVL C00159 BC00159 V=166.7  +MOVJ EC00159 VJ=100.00
SREFP 3 C00160 BC00160  +REFP EC00160
CALL JOB:SEARCH-R1-S13D
SET P062 P006
SFTON3D P062
SMOVL C00161 BC00161 V=166.7  +MOVJ EC00161
SREFP 3 C00162 BC00162  +REFP EC00162
CALL JOB:SEARCH-R1-S13D
SET P062 P006
SFTON3D P062
SMOVL C00163 BC00163 V=166.7  +MOVJ EC00163
SREFP 3 C00164 BC00164  +REFP EC00164
CALL JOB:SEARCH-R1-S13D
SET P062 P006
SFTON3D P062
SMOVL C00165 BC00165 V=166.7  +MOVJ EC00165
MOVL C00166 BC00166 V=666.7  +MOVJ EC00166 VJ=100.00
MOVL C00167 BC00167 V=666.7  +MOVJ EC00167 VJ=100.00
MOVL C00168 BC00168 V=166.7  +MOVJ EC00168 VJ=100.00
SREFP 3 C00169 BC00169  +REFP EC00169
CALL JOB:SEARCH-R1-S13D
SET P065 P006
SFTON3D P065
SMOVL C00170 BC00170 V=166.7  +MOVJ EC00170
SREFP 3 C00171 BC00171  +REFP EC00171
CALL JOB:SEARCH-R1-S13D
SET P065 P006
SFTON3D P065
SMOVL C00172 BC00172 V=166.7  +MOVJ EC00172
SMOVL C00173 BC00173 V=166.7  +MOVJ EC00173
SREFP 3 C00174 BC00174  +REFP EC00174
CALL JOB:SEARCH-R1-S13D
SET P065 P006
SFTON3D P065
SMOVL C00175 BC00175 V=166.7  +MOVJ EC00175
MOVL C00176 BC00176 V=666.7  +MOVJ EC00176 VJ=100.00
MOVL C00177 BC00177 V=166.7  +MOVJ EC00177 VJ=100.00
SREFP 3 C00178 BC00178  +REFP EC00178
CALL JOB:SEARCH-R1-S13D
SET P064 P006
SFTON3D P064
SMOVL C00179 BC00179 V=166.7  +MOVJ EC00179
SREFP 3 C00180 BC00180  +REFP EC00180
CALL JOB:SEARCH-R1-S13D
SET P064 P006
SFTON3D P064
SMOVL C00181 BC00181 V=166.7  +MOVJ EC00181
SMOVL C00182 BC00182 V=166.7  +MOVJ EC00182
SREFP 3 C00183 BC00183  +REFP EC00183
CALL JOB:SEARCH-R1-S13D
SET P064 P006
SFTON3D P064
SMOVL C00184 BC00184 V=166.7  +MOVJ EC00184
SFTOF3D
MOVL C00185 BC00185 V=666.7  +MOVJ EC00185 VJ=100.00
MOVL C00186 BC00186 V=666.7  +MOVJ EC00186 VJ=100.00
MOVJ C00187 BC00187 VJ=100.00  +MOVJ EC00187 VJ=100.00
MOVJ C00188 BC00188 VJ=100.00  +MOVJ EC00188 VJ=100.00
'Path S3853
SFTOF3D
MOVJ C00189 BC00189 VJ=100.00  +MOVJ EC00189 VJ=100.00
MOVL C00190 BC00190 V=800.0  +MOVJ EC00190 VJ=100.00
SMOVL C00191 BC00191 V=166.7  +MOVJ EC00191
SREFP 3 C00192 BC00192  +REFP EC00192
CALL JOB:SEARCH-R1-S13D
SET P023 P006
SFTON3D P023
SMOVL C00193 BC00193 V=166.7  +MOVJ EC00193
SREFP 3 C00194 BC00194  +REFP EC00194
CALL JOB:SEARCH-R1-S13D
SET P023 P006
SFTON3D P023
SMOVL C00195 BC00195 V=166.7  +MOVJ EC00195
SREFP 3 C00196 BC00196  +REFP EC00196
CALL JOB:SEARCH-R1-S13D
SET P023 P006
SFTON3D P023
SMOVL C00197 BC00197 V=166.7  +MOVJ EC00197
MOVL C00198 BC00198 V=800.0  +MOVJ EC00198 VJ=100.00
MOVL C00199 BC00199 V=1000.0  +MOVJ EC00199 VJ=100.00
'EndPath S3853
'Path S4665
SFTOF3D
MOVJ C00200 BC00200 VJ=100.00  +MOVJ EC00200 VJ=100.00
MOVL C00201 BC00201 V=800.0  +MOVJ EC00201 VJ=100.00
SMOVL C00202 BC00202 V=166.7  +MOVJ EC00202
SREFP 3 C00203 BC00203  +REFP EC00203
CALL JOB:SEARCH-R1-S13D
SET P024 P006
SFTON3D P024
SMOVL C00204 BC00204 V=166.7  +MOVJ EC00204
SREFP 3 C00205 BC00205  +REFP EC00205
CALL JOB:SEARCH-R1-S13D
SET P024 P006
SFTON3D P024
SMOVL C00206 BC00206 V=166.7  +MOVJ EC00206
MOVL C00207 BC00207 V=800.0  +MOVJ EC00207 VJ=100.00
MOVL C00208 BC00208 V=1000.0  +MOVJ EC00208 VJ=100.00
'EndPath S4665
MOVJ C00209 BC00209 VJ=100.00  +MOVJ EC00209 VJ=100.00
MOVJ C00210 BC00210 VJ=100.00  +MOVJ EC00210 VJ=100.00
'Path S3854
SFTOF3D
MOVJ C00211 BC00211 VJ=100.00  +MOVJ EC00211 VJ=100.00
MOVL C00212 BC00212 V=800.0  +MOVJ EC00212 VJ=100.00
SMOVL C00213 BC00213 V=166.7  +MOVJ EC00213
SREFP 3 C00214 BC00214  +REFP EC00214
CALL JOB:SEARCH-R1-S13D
SET P025 P006
SFTON3D P025
SMOVL C00215 BC00215 V=166.7  +MOVJ EC00215
SREFP 3 C00216 BC00216  +REFP EC00216
CALL JOB:SEARCH-R1-S13D
SET P025 P006
SFTON3D P025
SMOVL C00217 BC00217 V=166.7  +MOVJ EC00217
MOVL C00218 BC00218 V=800.0  +MOVJ EC00218 VJ=100.00
MOVL C00219 BC00219 V=1000.0  +MOVJ EC00219 VJ=100.00
'EndPath S3854
'Path S3855
SFTOF3D
MOVJ C00220 BC00220 VJ=100.00  +MOVJ EC00220 VJ=100.00
MOVL C00221 BC00221 V=800.0  +MOVJ EC00221 VJ=100.00
SMOVL C00222 BC00222 V=166.7  +MOVJ EC00222
SREFP 3 C00223 BC00223  +REFP EC00223
CALL JOB:SEARCH-R1-S13D
SET P026 P006
SFTON3D P026
SMOVL C00224 BC00224 V=166.7  +MOVJ EC00224
SREFP 3 C00225 BC00225  +REFP EC00225
CALL JOB:SEARCH-R1-S13D
SET P026 P006
SFTON3D P026
SMOVL C00226 BC00226 V=166.7  +MOVJ EC00226
MOVL C00227 BC00227 V=800.0  +MOVJ EC00227 VJ=100.00
MOVL C00228 BC00228 V=1000.0  +MOVJ EC00228 VJ=100.00
'EndPath S3855
MOVJ C00229 BC00229 VJ=100.00  +MOVJ EC00229 VJ=100.00
MOVJ C00230 BC00230 VJ=100.00  +MOVJ EC00230 VJ=100.00
'Up
MOVJ C00231 BC00231 VJ=100.00  +MOVJ EC00231 VJ=100.00
MOVJ C00232 BC00232 VJ=100.00  +MOVJ EC00232 VJ=100.00
'Path S3856
SFTOF3D
MOVJ C00233 BC00233 VJ=100.00  +MOVJ EC00233 VJ=100.00
MOVL C00234 BC00234 V=800.0  +MOVJ EC00234 VJ=100.00
SMOVL C00235 BC00235 V=166.7  +MOVJ EC00235
SREFP 3 C00236 BC00236  +REFP EC00236
CALL JOB:SEARCH-R1-S13D
SET P031 P006
SFTON3D P031
SMOVL C00237 BC00237 V=166.7  +MOVJ EC00237
SMOVL C00238 BC00238 V=166.7  +MOVJ EC00238
SREFP 3 C00239 BC00239  +REFP EC00239
CALL JOB:SEARCH-R1-S13D
SET P031 P006
SFTON3D P031
SMOVL C00240 BC00240 V=166.7  +MOVJ EC00240
SMOVL C00241 BC00241 V=166.7  +MOVJ EC00241
SREFP 3 C00242 BC00242  +REFP EC00242
CALL JOB:SEARCH-R1-S13D
SET P031 P006
SFTON3D P031
SMOVL C00243 BC00243 V=166.7  +MOVJ EC00243
MOVL C00244 BC00244 V=800.0  +MOVJ EC00244 VJ=100.00
MOVL C00245 BC00245 V=1000.0  +MOVJ EC00245 VJ=100.00
'EndPath S3856
MOVJ C00246 BC00246 VJ=100.00  +MOVJ EC00246 VJ=100.00
'Path S4666
SFTOF3D
MOVJ C00247 BC00247 VJ=100.00  +MOVJ EC00247 VJ=100.00
MOVL C00248 BC00248 V=800.0  +MOVJ EC00248 VJ=100.00
SMOVL C00249 BC00249 V=166.7  +MOVJ EC00249
SREFP 3 C00250 BC00250  +REFP EC00250
CALL JOB:SEARCH-R1-S13D
SET P032 P006
SFTON3D P032
SMOVL C00251 BC00251 V=166.7  +MOVJ EC00251
SMOVL C00252 BC00252 V=166.7  +MOVJ EC00252
SREFP 3 C00253 BC00253  +REFP EC00253
CALL JOB:SEARCH-R1-S13D
SET P032 P006
SFTON3D P032
SMOVL C00254 BC00254 V=166.7  +MOVJ EC00254
SMOVL C00255 BC00255 V=166.7  +MOVJ EC00255
SREFP 3 C00256 BC00256  +REFP EC00256
CALL JOB:SEARCH-R1-S13D
SET P032 P006
SFTON3D P032
SMOVL C00257 BC00257 V=166.7  +MOVJ EC00257
MOVL C00258 BC00258 V=800.0  +MOVJ EC00258 VJ=100.00
MOVL C00259 BC00259 V=1000.0  +MOVJ EC00259 VJ=100.00
'EndPath S4666
MOVJ C00260 BC00260 VJ=100.00  +MOVJ EC00260 VJ=100.00
'Path S3857
SFTOF3D
MOVJ C00261 BC00261 VJ=100.00  +MOVJ EC00261 VJ=100.00
MOVL C00262 BC00262 V=800.0  +MOVJ EC00262 VJ=100.00
SMOVL C00263 BC00263 V=166.7  +MOVJ EC00263
SREFP 3 C00264 BC00264  +REFP EC00264
CALL JOB:SEARCH-R1-S13D
SET P033 P006
SFTON3D P033
SMOVL C00265 BC00265 V=166.7  +MOVJ EC00265
SMOVL C00266 BC00266 V=166.7  +MOVJ EC00266
SREFP 3 C00267 BC00267  +REFP EC00267
CALL JOB:SEARCH-R1-S13D
SET P033 P006
SFTON3D P033
SMOVL C00268 BC00268 V=166.7  +MOVJ EC00268
SMOVL C00269 BC00269 V=166.7  +MOVJ EC00269
SREFP 3 C00270 BC00270  +REFP EC00270
CALL JOB:SEARCH-R1-S13D
SET P033 P006
SFTON3D P033
SMOVL C00271 BC00271 V=166.7  +MOVJ EC00271
MOVL C00272 BC00272 V=800.0  +MOVJ EC00272 VJ=100.00
MOVL C00273 BC00273 V=1000.0  +MOVJ EC00273 VJ=100.00
MOVL C00274 BC00274 V=1000.0  +MOVJ EC00274 VJ=100.00
'EndPath S3857
MOVJ C00275 BC00275 VJ=100.00  +MOVJ EC00275 VJ=100.00
'Path S4667
SFTOF3D
MOVJ C00276 BC00276 VJ=100.00  +MOVJ EC00276 VJ=100.00
MOVL C00277 BC00277 V=800.0  +MOVJ EC00277 VJ=100.00
SMOVL C00278 BC00278 V=166.7  +MOVJ EC00278
SREFP 3 C00279 BC00279  +REFP EC00279
CALL JOB:SEARCH-R1-S13D
SET P034 P006
SFTON3D P034
SMOVL C00280 BC00280 V=166.7  +MOVJ EC00280
SMOVL C00281 BC00281 V=166.7  +MOVJ EC00281
SREFP 3 C00282 BC00282  +REFP EC00282
CALL JOB:SEARCH-R1-S13D
SET P034 P006
SFTON3D P034
SMOVL C00283 BC00283 V=166.7  +MOVJ EC00283
SMOVL C00284 BC00284 V=166.7  +MOVJ EC00284
SREFP 3 C00285 BC00285  +REFP EC00285
CALL JOB:SEARCH-R1-S13D
SET P034 P006
SFTON3D P034
SMOVL C00286 BC00286 V=166.7  +MOVJ EC00286
MOVL C00287 BC00287 V=800.0  +MOVJ EC00287 VJ=100.00
MOVL C00288 BC00288 V=1000.0  +MOVJ EC00288 VJ=100.00
MOVL C00289 BC00289 V=1000.0  +MOVJ EC00289 VJ=100.00
'EndPath S4667
MOVJ C00290 BC00290 VJ=100.00  +MOVJ EC00290 VJ=100.00
'Path S4668
SFTOF3D
MOVJ C00291 BC00291 VJ=100.00  +MOVJ EC00291 VJ=100.00
MOVL C00292 BC00292 V=800.0  +MOVJ EC00292 VJ=100.00
SMOVL C00293 BC00293 V=166.7  +MOVJ EC00293
SREFP 3 C00294 BC00294  +REFP EC00294
CALL JOB:SEARCH-R1-S13D
SET P035 P006
SFTON3D P035
SMOVL C00295 BC00295 V=166.7  +MOVJ EC00295
SMOVL C00296 BC00296 V=166.7  +MOVJ EC00296
SREFP 3 C00297 BC00297  +REFP EC00297
CALL JOB:SEARCH-R1-S13D
SET P035 P006
SFTON3D P035
SMOVL C00298 BC00298 V=166.7  +MOVJ EC00298
SMOVL C00299 BC00299 V=166.7  +MOVJ EC00299
SREFP 3 C00300 BC00300  +REFP EC00300
CALL JOB:SEARCH-R1-S13D
SET P035 P006
SFTON3D P035
SMOVL C00301 BC00301 V=166.7  +MOVJ EC00301
MOVL C00302 BC00302 V=800.0  +MOVJ EC00302 VJ=100.00
MOVL C00303 BC00303 V=1000.0  +MOVJ EC00303 VJ=100.00
'EndPath S4668
MOVJ C00304 BC00304 VJ=100.00  +MOVJ EC00304 VJ=100.00
'Path S4669
SFTOF3D
MOVJ C00305 BC00305 VJ=100.00  +MOVJ EC00305 VJ=100.00
MOVL C00306 BC00306 V=800.0  +MOVJ EC00306 VJ=100.00
SMOVL C00307 BC00307 V=166.7  +MOVJ EC00307
SREFP 3 C00308 BC00308  +REFP EC00308
CALL JOB:SEARCH-R1-S13D
SET P036 P006
SFTON3D P036
SMOVL C00309 BC00309 V=166.7  +MOVJ EC00309
SMOVL C00310 BC00310 V=166.7  +MOVJ EC00310
SREFP 3 C00311 BC00311  +REFP EC00311
CALL JOB:SEARCH-R1-S13D
SET P036 P006
SFTON3D P036
SMOVL C00312 BC00312 V=166.7  +MOVJ EC00312
SMOVL C00313 BC00313 V=166.7  +MOVJ EC00313
SREFP 3 C00314 BC00314  +REFP EC00314
CALL JOB:SEARCH-R1-S13D
SET P036 P006
SFTON3D P036
SMOVL C00315 BC00315 V=166.7  +MOVJ EC00315
MOVL C00316 BC00316 V=800.0  +MOVJ EC00316 VJ=100.00
MOVL C00317 BC00317 V=1000.0  +MOVJ EC00317 VJ=100.00
'EndPath S4669
MOVJ C00318 BC00318 VJ=100.00  +MOVJ EC00318 VJ=100.00
'Path S3859
SFTOF3D
MOVJ C00319 BC00319 VJ=100.00  +MOVJ EC00319 VJ=100.00
MOVL C00320 BC00320 V=800.0  +MOVJ EC00320 VJ=100.00
SMOVL C00321 BC00321 V=166.7  +MOVJ EC00321
SREFP 3 C00322 BC00322  +REFP EC00322
CALL JOB:SEARCH-R1-S13D
SET P037 P006
SFTON3D P037
SMOVL C00323 BC00323 V=166.7  +MOVJ EC00323
SMOVL C00324 BC00324 V=166.7  +MOVJ EC00324
SREFP 3 C00325 BC00325  +REFP EC00325
CALL JOB:SEARCH-R1-S13D
SET P037 P006
SFTON3D P037
SMOVL C00326 BC00326 V=166.7  +MOVJ EC00326
SMOVL C00327 BC00327 V=166.7  +MOVJ EC00327
SREFP 3 C00328 BC00328  +REFP EC00328
CALL JOB:SEARCH-R1-S13D
SET P037 P006
SFTON3D P037
SMOVL C00329 BC00329 V=166.7  +MOVJ EC00329
MOVL C00330 BC00330 V=800.0  +MOVJ EC00330 VJ=100.00
MOVL C00331 BC00331 V=1000.0  +MOVJ EC00331 VJ=100.00
'EndPath S3859
MOVJ C00332 BC00332 VJ=100.00  +MOVJ EC00332 VJ=100.00
'Path S4670
SFTOF3D
MOVJ C00333 BC00333 VJ=100.00  +MOVJ EC00333 VJ=100.00
MOVL C00334 BC00334 V=800.0  +MOVJ EC00334 VJ=100.00
SMOVL C00335 BC00335 V=166.7  +MOVJ EC00335
SREFP 3 C00336 BC00336  +REFP EC00336
CALL JOB:SEARCH-R1-S13D
SET P038 P006
SFTON3D P038
SMOVL C00337 BC00337 V=166.7  +MOVJ EC00337
SMOVL C00338 BC00338 V=166.7  +MOVJ EC00338
SREFP 3 C00339 BC00339  +REFP EC00339
CALL JOB:SEARCH-R1-S13D
SET P038 P006
SFTON3D P038
SMOVL C00340 BC00340 V=166.7  +MOVJ EC00340
SMOVL C00341 BC00341 V=166.7  +MOVJ EC00341
SREFP 3 C00342 BC00342  +REFP EC00342
CALL JOB:SEARCH-R1-S13D
SET P038 P006
SFTON3D P038
SMOVL C00343 BC00343 V=166.7  +MOVJ EC00343
MOVL C00344 BC00344 V=800.0  +MOVJ EC00344 VJ=100.00
MOVL C00345 BC00345 V=1000.0  +MOVJ EC00345 VJ=100.00
'EndPath S4670
MOVJ C00346 BC00346 VJ=100.00  +MOVJ EC00346 VJ=100.00
'Path S3860
SFTOF3D
MOVJ C00347 BC00347 VJ=100.00  +MOVJ EC00347 VJ=100.00
MOVL C00348 BC00348 V=800.0  +MOVJ EC00348 VJ=100.00
SMOVL C00349 BC00349 V=166.7  +MOVJ EC00349
SREFP 3 C00350 BC00350  +REFP EC00350
CALL JOB:SEARCH-R1-S13D
SET P039 P006
SFTON3D P039
SMOVL C00351 BC00351 V=166.7  +MOVJ EC00351
SMOVL C00352 BC00352 V=166.7  +MOVJ EC00352
SREFP 3 C00353 BC00353  +REFP EC00353
CALL JOB:SEARCH-R1-S13D
SET P039 P006
SFTON3D P039
SMOVL C00354 BC00354 V=166.7  +MOVJ EC00354
SMOVL C00355 BC00355 V=166.7  +MOVJ EC00355
SREFP 3 C00356 BC00356  +REFP EC00356
CALL JOB:SEARCH-R1-S13D
SET P039 P006
SFTON3D P039
SMOVL C00357 BC00357 V=166.7  +MOVJ EC00357
MOVL C00358 BC00358 V=800.0  +MOVJ EC00358 VJ=100.00
MOVL C00359 BC00359 V=1000.0  +MOVJ EC00359 VJ=100.00
'EndPath S3860
'Path S4671
SFTOF3D
MOVJ C00360 BC00360 VJ=100.00  +MOVJ EC00360 VJ=100.00
MOVL C00361 BC00361 V=800.0  +MOVJ EC00361 VJ=100.00
SMOVL C00362 BC00362 V=166.7  +MOVJ EC00362
SREFP 3 C00363 BC00363  +REFP EC00363
CALL JOB:SEARCH-R1-S13D
SET P040 P006
SFTON3D P040
SMOVL C00364 BC00364 V=166.7  +MOVJ EC00364
SMOVL C00365 BC00365 V=166.7  +MOVJ EC00365
SREFP 3 C00366 BC00366  +REFP EC00366
CALL JOB:SEARCH-R1-S13D
SET P040 P006
SFTON3D P040
SMOVL C00367 BC00367 V=166.7  +MOVJ EC00367
MOVL C00368 BC00368 V=800.0  +MOVJ EC00368 VJ=100.00
MOVL C00369 BC00369 V=1000.0  +MOVJ EC00369 VJ=100.00
'EndPath S4671
'Path W3861
SFTOF3D
SFTON3D P039
MOVJ C00370 BC00370 VJ=100.00  +MOVJ EC00370 VJ=100.00
SMOVL C00371 BC00371 V=800.0  +MOVJ EC00371
SMOVL C00372 BC00372 V=166.7 PL=0  +MOVJ EC00372
MACRO1 MJ#(0) ARGF9
ARCON
SMOVL C00373 BC00373 V=7.5  +MOVJ EC00373
SFTON3D P040
SMOVL C00374 BC00374 V=7.5  +MOVJ EC00374
SMOVL C00375 BC00375 V=7.5  +MOVJ EC00375
ARCOF
SMOVL C00376 BC00376 V=800.0  +MOVJ EC00376
SMOVL C00377 BC00377 V=1000.0  +MOVJ EC00377
SFTOF3D
'EndPath W3861
MOVJ C00378 BC00378 VJ=100.00  +MOVJ EC00378 VJ=100.00
'Path W3862
SFTOF3D
SFTON3D P037
MOVJ C00379 BC00379 VJ=100.00  +MOVJ EC00379 VJ=100.00
MOVJ C00380 BC00380 VJ=100.00  +MOVJ EC00380 VJ=100.00
SMOVL C00381 BC00381 V=800.0  +MOVJ EC00381
SMOVL C00382 BC00382 V=166.7 PL=0  +MOVJ EC00382
MACRO1 MJ#(0) ARGF14
ARCON
SMOVL C00383 BC00383 V=10.0  +MOVJ EC00383
SMOVL C00384 BC00384 V=10.0  +MOVJ EC00384
SFTON3D P038
SMOVL C00385 BC00385 V=10.0  +MOVJ EC00385
SMOVL C00386 BC00386 V=10.0  +MOVJ EC00386
ARCOF
SMOVL C00387 BC00387 V=800.0  +MOVJ EC00387
SMOVL C00388 BC00388 V=1000.0  +MOVJ EC00388
SFTOF3D
'EndPath W3862
MOVJ C00389 BC00389 VJ=100.00  +MOVJ EC00389 VJ=100.00
MOVJ C00390 BC00390 VJ=100.00  +MOVJ EC00390 VJ=100.00
'Path W3863
SFTOF3D
SFTON3D P035
MOVJ C00391 BC00391 VJ=100.00  +MOVJ EC00391 VJ=100.00
MOVJ C00392 BC00392 VJ=100.00  +MOVJ EC00392 VJ=100.00
SMOVL C00393 BC00393 V=800.0  +MOVJ EC00393
SMOVL C00394 BC00394 V=166.7 PL=0  +MOVJ EC00394
ARCON
SMOVL C00395 BC00395 V=9.2  +MOVJ EC00395
SFTON3D P036
SMOVL C00396 BC00396 V=9.2  +MOVJ EC00396
SMOVL C00397 BC00397 V=9.2  +MOVJ EC00397
ARCOF
